KUKA KRL program: MyProgram_337().src

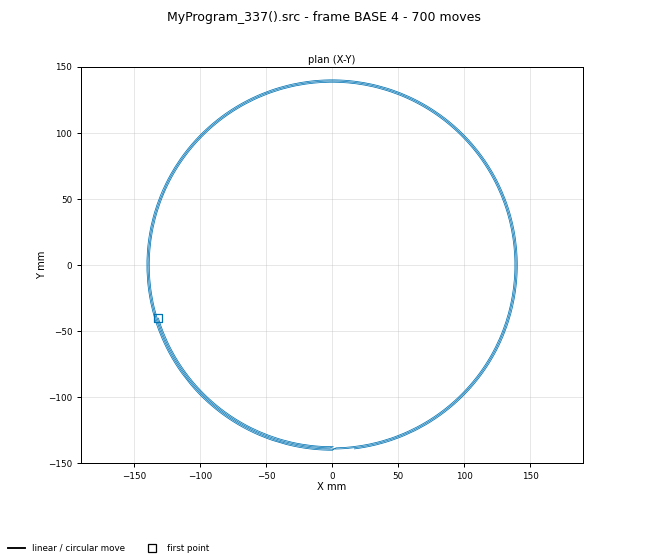
[picture p0: tool path of MyProgram_337().src in frame BASE 4, 700 of 700 moves have a stored position in this frame; points joined in program order, loops and branches not executed]
&ACCESS RVP
&REL 1
&PARAM TEMPLATE = C:\KRC\Roboter\Template\vorgabe
&PARAM EDITMASK = *
DEF MyProgram_337()
; ---- Setting reference (Base) ----
$BASE = BASE_DATA[4]

; --------------------------
; ---- Setting tool (TCP) ----
$TOOL = TOOL_DATA[3]
; --------------------------

$VEL.CP = VEL_APROX_PRINT
Startdeposition()
$VEL.CP = VEL_PRINT
LIN {X -131.5627,Y -40.1992,Z 190,A -156.4352,B 1.1423,C 0.1249,E1 0.9973,E2 249.9289} C_DIS
LIN {X -130.6707,Y -43.0129,Z 190,A -155.1283,B 1.1419,C 0.1281,E1 0.9985,E2 248.6121} C_DIS
LIN {X -129.6796,Y -45.9186,Z 190,A -153.4,B 1.1415,C 0.1315,E1 1.0001,E2 246.8238} C_DIS
LIN {X -127.8186,Y -50.8673,Z 190,A -150.9878,B 1.1409,C 0.1372,E1 1.0026,E2 244.3839} C_DIS
LIN {X -126.194,Y -54.7705,Z 190,A -149.1607,B 1.1403,C 0.1416,E1 1.0046,E2 242.5483} C_DIS
LIN {X -124.9534,Y -57.5445,Z 190,A -147.6737,B 1.14,C 0.1447,E1 1.0063,E2 241.0315} C_DIS
LIN {X -123.462,Y -60.6782,Z 190,A -146.0319,B 1.1395,C 0.1482,E1 1.0084,E2 239.3634} C_DIS
LIN {X -121.5451,Y -64.4341,Z 190,A -143.3556,B 1.139,C 0.1523,E1 1.0121,E2 236.5609} C_DIS
LIN {X -118.9555,Y -69.1002,Z 190,A -141.515,B 1.1383,C 0.1574,E1 1.0145,E2 234.7739} C_DIS
LIN {X -116.3723,Y -73.367,Z 190,A -139.2239,B 1.1376,C 0.162,E1 1.0179,E2 232.4537} C_DIS
LIN {X -113.9274,Y -77.1089,Z 190,A -137.1564,B 1.137,C 0.166,E1 1.0212,E2 230.3581} C_DIS
LIN {X -111.3595,Y -80.7731,Z 190,A -135.1136,B 1.1365,C 0.1699,E1 1.0245,E2 228.2907} C_DIS
LIN {X -108.6208,Y -84.4203,Z 190,A -132.998,B 1.1359,C 0.1736,E1 1.0282,E2 226.1454} C_DIS
LIN {X -105.7296,Y -88.0148,Z 190,A -130.861,B 1.1353,C 0.1773,E1 1.032,E2 223.9785} C_DIS
LIN {X -102.7599,Y -91.4648,Z 190,A -128.8416,B 1.1348,C 0.1808,E1 1.0358,E2 221.942} C_DIS
LIN {X -99.7983,Y -94.6873,Z 190,A -126.928,B 1.1343,C 0.1841,E1 1.0395,E2 220.0158} C_DIS
LIN {X -97.1901,Y -97.3623,Z 190,A -125.164,B 1.1338,C 0.1866,E1 1.043,E2 218.2226} C_DIS
LIN {X -94.7289,Y -99.7586,Z 190,A -123.479,B 1.1335,C 0.1888,E1 1.0465,E2 216.5018} C_DIS
LIN {X -90.9578,Y -103.2083,Z 190,A -121.3105,B 1.1329,C 0.1922,E1 1.0511,E2 214.3277} C_DIS
LIN {X -87.7491,Y -105.9496,Z 190,A -119.4335,B 1.1325,C 0.1947,E1 1.0552,E2 212.4338} C_DIS
LIN {X -84.3581,Y -108.669,Z 190,A -117.4741,B 1.1321,C 0.1972,E1 1.0595,E2 210.4532} C_DIS
LIN {X -80.6661,Y -111.4371,Z 190,A -115.4682,B 1.1316,C 0.1997,E1 1.0641,E2 208.4352} C_DIS
LIN {X -76.4637,Y -114.3615,Z 190,A -113.1651,B 1.1312,C 0.2022,E1 1.0695,E2 206.1076} C_DIS
LIN {X -72.9085,Y -116.6604,Z 190,A -111.1391,B 1.1309,C 0.2038,E1 1.0744,E2 204.0438} C_DIS
LIN {X -68.4116,Y -119.3531,Z 190,A -109.0245,B 1.1304,C 0.2063,E1 1.0795,E2 201.9387} C_DIS
LIN {X -64.6433,Y -121.4352,Z 190,A -107.1659,B 1.1301,C 0.208,E1 1.0842,E2 200.0705} C_DIS
LIN {X -61.1965,Y -123.2063,Z 190,A -105.6298,B 1.1298,C 0.2096,E1 1.088,E2 198.5452} C_DIS
LIN {X -57.9125,Y -124.7833,Z 190,A -104.2309,B 1.1295,C 0.2111,E1 1.0915,E2 197.1629} C_DIS
LIN {X -55.1219,Y -126.0421,Z 190,A -102.628,B 1.1295,C 0.2114,E1 1.0958,E2 195.5128} C_DIS
LIN {X -50.5791,Y -127.9339,Z 190,A -100.5694,B 1.1292,C 0.2128,E1 1.1011,E2 193.4524} C_DIS
LIN {X -47.9087,Y -128.9558,Z 190,A -99.21,B 1.1292,C 0.2132,E1 1.1048,E2 192.0684} C_DIS
LIN {X -43.7636,Y -130.4207,Z 190,A -97.4491,B 1.1289,C 0.2143,E1 1.1095,E2 190.3171} C_DIS
LIN {X -40.8951,Y -131.3497,Z 190,A -96.2332,B 1.1289,C 0.215,E1 1.1127,E2 189.1065} C_DIS
LIN {X -37.3559,Y -132.3985,Z 190,A -94.5915,B 1.1287,C 0.2153,E1 1.1172,E2 187.4493} C_DIS
LIN {X -33.9694,Y -133.3073,Z 190,A -93.1469,B 1.1287,C 0.2158,E1 1.1211,E2 186.0065} C_DIS
LIN {X -30.8122,Y -134.0724,Z 190,A -91.8493,B 1.1286,C 0.2163,E1 1.1247,E2 184.7163} C_DIS
LIN {X -26.9975,Y -134.8929,Z 190,A -89.6626,B 1.1288,C 0.2151,E1 1.1309,E2 182.4478} C_DIS
LIN {X -22.9337,Y -135.6426,Z 190,A -88.3319,B 1.1286,C 0.2163,E1 1.1345,E2 181.1729} C_DIS
LIN {X -16.4531,Y -136.5801,Z 190,A -85.5629,B 1.1286,C 0.2161,E1 1.1422,E2 178.3968} C_DIS
LIN {X -12.3209,Y -137.0166,Z 190,A -83.8051,B 1.1286,C 0.2158,E1 1.1472,E2 176.6343} C_DIS
LIN {X -8.3051,Y -137.3167,Z 190,A -82.2397,B 1.1286,C 0.2158,E1 1.1515,E2 175.0842} C_DIS
LIN {X -4.2325,Y -137.5031,Z 190,A -80.452,B 1.1288,C 0.2151,E1 1.1566,E2 173.2827} C_DIS
LIN {X 0.983,Y -137.5643,Z 190,A -78.8429,B 1.1286,C 0.2161,E1 1.1609,E2 171.7536} C_DIS
Enddeposition()
LIN {X 0.983,Y -137.5643,Z 190,A -78.843,B 1.1286,C 0.2161,E1 1.1609,E2 171.7538} C_DIS
Startdeposition()
$VEL.CP = VEL_PRINT
LIN {X -1.5333,Y -138.4601,Z 190,A -80.1965,B 1.1539,C 0.2192,E1 1.1826,E2 173.1713} C_DIS
LIN {X -4.6035,Y -138.392,Z 190,A -81.4508,B 1.1539,C 0.2195,E1 1.1791,E2 174.4239} C_DIS
LIN {X -8.8461,Y -138.184,Z 190,A -83.1886,B 1.1538,C 0.2199,E1 1.1742,E2 176.1597} C_DIS
LIN {X -12.4098,Y -137.9112,Z 190,A -84.6675,B 1.1538,C 0.2201,E1 1.17,E2 177.6394} C_DIS
LIN {X -15.5748,Y -137.5897,Z 190,A -85.981,B 1.1537,C 0.2202,E1 1.1663,E2 178.953} C_DIS
LIN {X -18.757,Y -137.1921,Z 190,A -87.3061,B 1.1537,C 0.2202,E1 1.1626,E2 180.2785} C_DIS
LIN {X -21.4733,Y -136.7914,Z 190,A -88.4926,B 1.1537,C 0.2204,E1 1.1593,E2 181.4726} C_DIS
LIN {X -25.1634,Y -136.1628,Z 190,A -90.0069,B 1.1537,C 0.2201,E1 1.1551,E2 182.9826} C_DIS
LIN {X -28.0039,Y -135.6054,Z 190,A -91.2463,B 1.1537,C 0.2201,E1 1.1517,E2 184.2285} C_DIS
LIN {X -31.6408,Y -134.8051,Z 190,A -92.7737,B 1.1538,C 0.2196,E1 1.1475,E2 185.7545} C_DIS
LIN {X -34.7188,Y -134.0445,Z 190,A -94.103,B 1.1538,C 0.2193,E1 1.1438,E2 187.0868} C_DIS
LIN {X -38.1008,Y -133.1236,Z 190,A -95.5818,B 1.154,C 0.2188,E1 1.1398,E2 188.5702} C_DIS
LIN {X -41.3291,Y -132.157,Z 190,A -97.0049,B 1.154,C 0.2183,E1 1.136,E2 189.9978} C_DIS
LIN {X -44.5521,Y -131.1056,Z 190,A -98.4415,B 1.1542,C 0.2176,E1 1.1321,E2 191.4398} C_DIS
LIN {X -47.7339,Y -129.9807,Z 190,A -99.8757,B 1.1543,C 0.2169,E1 1.1283,E2 192.8798} C_DIS
LIN {X -50.9696,Y -128.7465,Z 190,A -101.3517,B 1.1545,C 0.2161,E1 1.1244,E2 194.3623} C_DIS
LIN {X -54.0161,Y -127.4974,Z 190,A -102.7597,B 1.1546,C 0.2152,E1 1.1207,E2 195.7771} C_DIS
LIN {X -57.0709,Y -126.1589,Z 190,A -104.2036,B 1.1548,C 0.2142,E1 1.117,E2 197.2304} C_DIS
LIN {X -60.475,Y -124.5646,Z 190,A -105.8075,B 1.155,C 0.213,E1 1.1129,E2 198.8416} C_DIS
LIN {X -63.5979,Y -122.9995,Z 190,A -107.3149,B 1.1553,C 0.2118,E1 1.1091,E2 200.3582} C_DIS
LIN {X -66.31,Y -121.558,Z 190,A -108.7108,B 1.1555,C 0.2107,E1 1.1056,E2 201.7721} C_DIS
LIN {X -69.755,Y -119.6152,Z 190,A -110.3598,B 1.1558,C 0.209,E1 1.1015,E2 203.4232} C_DIS
LIN {X -72.6195,Y -117.8975,Z 190,A -111.8361,B 1.156,C 0.2076,E1 1.098,E2 204.913} C_DIS
LIN {X -76.1626,Y -115.64,Z 190,A -113.7142,B 1.1564,C 0.2057,E1 1.0935,E2 206.8112} C_DIS
LIN {X -79.8624,Y -113.1166,Z 190,A -115.672,B 1.1568,C 0.2035,E1 1.0889,E2 208.784} C_DIS
LIN {X -83.039,Y -110.8065,Z 190,A -117.3467,B 1.1571,C 0.2013,E1 1.0851,E2 210.4658} C_DIS
LIN {X -86.2373,Y -108.3351,Z 190,A -119.2008,B 1.1575,C 0.1991,E1 1.0809,E2 212.3457} C_DIS
LIN {X -89.3427,Y -105.7896,Z 190,A -120.9923,B 1.1579,C 0.1968,E1 1.077,E2 214.1555} C_DIS
LIN {X -92.7012,Y -102.8593,Z 190,A -122.8956,B 1.1584,C 0.1939,E1 1.073,E2 216.067} C_DIS
LIN {X -95.3316,Y -100.4262,Z 190,A -124.4946,B 1.1588,C 0.1915,E1 1.0697,E2 217.6824} C_DIS
LIN {X -97.9121,Y -97.9121,Z 190,A -126.1074,B 1.1592,C 0.1891,E1 1.0664,E2 219.3123} C_DIS
LIN {X -100.6879,Y -95.0542,Z 190,A -127.9781,B 1.1597,C 0.1863,E1 1.0628,E2 221.2139} C_DIS
LIN {X -103.4567,Y -92.034,Z 190,A -129.8673,B 1.1601,C 0.1833,E1 1.0592,E2 223.13} C_DIS
LIN {X -106.4321,Y -88.5758,Z 190,A -131.9282,B 1.1607,C 0.1797,E1 1.0554,E2 225.2148} C_DIS
LIN {X -109.1582,Y -85.1941,Z 190,A -133.7748,B 1.1612,C 0.1761,E1 1.0521,E2 227.0679} C_DIS
LIN {X -111.328,Y -82.3386,Z 190,A -135.4036,B 1.1617,C 0.1732,E1 1.0494,E2 228.7166} C_DIS
LIN {X -113.257,Y -79.6633,Z 190,A -136.9417,B 1.1621,C 0.1703,E1 1.0468,E2 230.2784} C_DIS
LIN {X -115.4099,Y -76.5122,Z 190,A -138.6491,B 1.1626,C 0.167,E1 1.0441,E2 232.0032} C_DIS
LIN {X -117.3303,Y -73.5334,Z 190,A -140.3787,B 1.163,C 0.1638,E1 1.0415,E2 233.7687} C_DIS
LIN {X -119.6061,Y -69.7705,Z 190,A -142.2935,B 1.1636,C 0.1597,E1 1.0387,E2 235.6961} C_DIS
LIN {X -121.3495,Y -66.6923,Z 190,A -143.9218,B 1.1641,C 0.1563,E1 1.0365,E2 237.3465} C_DIS
LIN {X -122.9093,Y -63.7697,Z 190,A -145.4555,B 1.1645,C 0.1531,E1 1.0344,E2 238.9021} C_DIS
LIN {X -124.3492,Y -60.9117,Z 190,A -146.9699,B 1.1649,C 0.1499,E1 1.0325,E2 240.442} C_DIS
LIN {X -126.0443,Y -57.3271,Z 190,A -148.7649,B 1.1654,C 0.1459,E1 1.0304,E2 242.2575} C_DIS
LIN {X -127.4383,Y -54.1575,Z 190,A -150.3709,B 1.1659,C 0.1424,E1 1.0286,E2 243.8864} C_DIS
LIN {X -128.7334,Y -51.0022,Z 190,A -151.9557,B 1.1663,C 0.1388,E1 1.0269,E2 245.4942} C_DIS
LIN {X -129.9689,Y -47.7667,Z 190,A -153.5679,B 1.1667,C 0.1351,E1 1.0253,E2 247.13} C_DIS
LIN {X -131.0942,Y -44.585,Z 190,A -155.1384,B 1.1671,C 0.1315,E1 1.0238,E2 248.7233} C_DIS
LIN {X -132.157,Y -41.3291,Z 190,A -156.7397,B 1.1676,C 0.1277,E1 1.0224,E2 250.3487} C_DIS
LIN {X -132.9702,Y -38.6248,Z 190,A -158.0672,B 1.1679,C 0.1246,E1 1.0214,E2 251.6969} C_DIS
LIN {X -133.9972,Y -34.9033,Z 190,A -159.8584,B 1.1683,C 0.1203,E1 1.02,E2 253.5133} C_DIS
LIN {X -134.6974,Y -32.0879,Z 190,A -161.233,B 1.1687,C 0.117,E1 1.0191,E2 254.9104} C_DIS
LIN {X -135.4719,Y -28.6461,Z 190,A -162.8891,B 1.1691,C 0.113,E1 1.0181,E2 256.5918} C_DIS
LIN {X -136.135,Y -25.311,Z 190,A -164.4774,B 1.1694,C 0.1091,E1 1.0173,E2 258.2034} C_DIS
LIN {X -136.7119,Y -21.9868,Z 190,A -166.0584,B 1.1698,C 0.1052,E1 1.0165,E2 259.8081} C_DIS
LIN {X -137.3216,Y -17.7691,Z 190,A -168.1258,B 1.1702,C 0.1002,E1 1.0157,E2 261.9143} C_DIS
LIN {X -137.7568,Y -14.0223,Z 190,A -169.8359,B 1.1706,C 0.0958,E1 1.0152,E2 263.6432} C_DIS
LIN {X -138.0416,Y -10.8667,Z 190,A -171.3266,B 1.1709,C 0.0921,E1 1.0148,E2 265.1566} C_DIS
LIN {X -138.2526,Y -7.7319,Z 190,A -172.8055,B 1.1712,C 0.0884,E1 1.0146,E2 266.658} C_DIS
LIN {X -138.3726,Y -5.1056,Z 190,A -174.0489,B 1.1714,C 0.0853,E1 1.0144,E2 267.9209} C_DIS
LIN {X -138.4596,Y -1.5648,Z 190,A -175.7119,B 1.1717,C 0.0811,E1 1.0144,E2 269.6085} C_DIS
LIN {X -138.4606,Y 1.4676,Z 190,A -177.1471,B 1.172,C 0.0775,E1 1.0144,E2 271.0662} C_DIS
LIN {X -138.3915,Y 4.6201,Z 190,A -178.6333,B 1.1722,C 0.0737,E1 1.0144,E2 272.5749} C_DIS
LIN {X -138.2526,Y 7.7319,Z 190,A 179.8943,B 1.1724,C 0.0701,E1 1.0147,E2 274.0701} C_DIS
LIN {X -137.9596,Y 11.8371,Z 190,A 177.8799,B 1.1727,C 0.0651,E1 1.0151,E2 276.1229} C_DIS
LIN {X -137.5897,Y 15.5748,Z 190,A 176.1754,B 1.1729,C 0.0607,E1 1.0156,E2 277.8456} C_DIS
LIN {X -137.1921,Y 18.757,Z 190,A 174.6616,B 1.1731,C 0.057,E1 1.0162,E2 279.3821} C_DIS
LIN {X -136.7119,Y 21.9868,Z 190,A 173.1212,B 1.1733,C 0.0531,E1 1.0168,E2 280.9455} C_DIS
LIN {X -136.222,Y 24.8327,Z 190,A 171.7669,B 1.1735,C 0.0498,E1 1.0175,E2 282.319} C_DIS
LIN {X -135.5217,Y 28.4151,Z 190,A 170.0405,B 1.1736,C 0.0456,E1 1.0185,E2 284.0714} C_DIS
LIN {X -134.8051,Y 31.6408,Z 190,A 168.4855,B 1.1738,C 0.0418,E1 1.0195,E2 285.6489} C_DIS
LIN {X -134.0144,Y 34.8374,Z 190,A 166.9367,B 1.1739,C 0.038,E1 1.0205,E2 287.22} C_DIS
LIN {X -133.2721,Y 37.5697,Z 190,A 165.6011,B 1.174,C 0.0348,E1 1.0216,E2 288.5749} C_DIS
LIN {X -132.157,Y 41.3291,Z 190,A 163.7687,B 1.1741,C 0.0304,E1 1.0231,E2 290.4322} C_DIS
LIN {X -131.1056,Y 44.5521,Z 190,A 162.1808,B 1.1742,C 0.0267,E1 1.0245,E2 292.0419} C_DIS
LIN {X -130.095,Y 47.4168,Z 190,A 160.7715,B 1.1742,C 0.0234,E1 1.0258,E2 293.4689} C_DIS
LIN {X -128.8741,Y 50.6414,Z 190,A 159.1246,B 1.1744,C 0.0196,E1 1.0275,E2 295.1416} C_DIS
LIN {X -127.4383,Y 54.1575,Z 190,A 157.3795,B 1.1744,C 0.0156,E1 1.0294,E2 296.9069} C_DIS
LIN {X -126.0443,Y 57.3271,Z 190,A 155.7686,B 1.1744,C 0.012,E1 1.0313,E2 298.5384} C_DIS
LIN {X -124.5646,Y 60.475,Z 190,A 154.1532,B 1.1744,C 0.0084,E1 1.0332,E2 300.174} C_DIS
LIN {X -122.9995,Y 63.5979,Z 190,A 152.5345,B 1.1745,C 0.0049,E1 1.0353,E2 301.8125} C_DIS
LIN {X -121.3617,Y 66.6699,Z 190,A 150.9217,B 1.1745,C 0.0014,E1 1.0375,E2 303.4449} C_DIS
LIN {X -119.6152,Y 69.755,Z 190,A 149.2906,B 1.1745,C -0.002,E1 1.0398,E2 305.0947} C_DIS
LIN {X -117.6028,Y 73.0955,Z 190,A 147.4279,B 1.1745,C -0.0057,E1 1.0426,E2 306.9857} C_DIS
LIN {X -115.4099,Y 76.5122,Z 190,A 145.6313,B 1.1745,C -0.0094,E1 1.0453,E2 308.7951} C_DIS
LIN {X -113.4086,Y 79.4483,Z 190,A 144.0046,B 1.1745,C -0.0126,E1 1.0479,E2 310.4392} C_DIS
LIN {X -111.3388,Y 82.3239,Z 190,A 142.3848,B 1.1745,C -0.0157,E1 1.0507,E2 312.0761} C_DIS
LIN {X -108.8631,Y 85.5697,Z 190,A 140.465,B 1.1744,C -0.0192,E1 1.054,E2 314.0217} C_DIS
LIN {X -106.3646,Y 88.6574,Z 190,A 138.7225,B 1.1744,C -0.0224,E1 1.0571,E2 315.7747} C_DIS
LIN {X -104.0496,Y 91.3631,Z 190,A 137.1107,B 1.1742,C -0.0253,E1 1.0601,E2 317.4016} C_DIS
LIN {X -101.6514,Y 94.0241,Z 190,A 135.4942,B 1.1742,C -0.028,E1 1.0632,E2 319.0328} C_DIS
LIN {X -99.1712,Y 96.6366,Z 190,A 133.7491,B 1.1742,C -0.0306,E1 1.0666,E2 320.8063} C_DIS
LIN {X -95.9927,Y 99.7946,Z 190,A 131.8639,B 1.174,C -0.0339,E1 1.0704,E2 322.6938} C_DIS
LIN {X -93.3781,Y 102.2453,Z 190,A 130.2623,B 1.174,C -0.0363,E1 1.0738,E2 324.3082} C_DIS
LIN {X -90.7025,Y 104.6261,Z 190,A 128.6684,B 1.1739,C -0.0387,E1 1.0771,E2 325.914} C_DIS
LIN {X -87.7038,Y 107.1514,Z 190,A 126.8337,B 1.1739,C -0.041,E1 1.0812,E2 327.7719} C_DIS
LIN {X -84.4742,Y 109.7163,Z 190,A 125.1008,B 1.1737,C -0.0435,E1 1.085,E2 329.5067} C_DIS
LIN {X -81.8311,Y 111.7008,Z 190,A 123.6073,B 1.1737,C -0.0454,E1 1.0884,E2 331.0137} C_DIS
LIN {X -78.7334,Y 113.9061,Z 190,A 121.8818,B 1.1736,C -0.0473,E1 1.0924,E2 332.7555} C_DIS
LIN {X -75.0431,Y 116.3704,Z 190,A 120.0271,B 1.1735,C -0.0496,E1 1.0968,E2 334.6112} C_DIS
LIN {X -72.0291,Y 118.2598,Z 190,A 118.4772,B 1.1735,C -0.0513,E1 1.1005,E2 336.169} C_DIS
LIN {X -69.0081,Y 120.0476,Z 190,A 116.9506,B 1.1733,C -0.0528,E1 1.1042,E2 337.7031} C_DIS
LIN {X -65.5833,Y 121.9516,Z 190,A 115.1729,B 1.1733,C -0.0543,E1 1.1087,E2 339.4974} C_DIS
LIN {X -62.0716,Y 123.7765,Z 190,A 113.5443,B 1.1732,C -0.0559,E1 1.1127,E2 341.1241} C_DIS
LIN {X -59.317,Y 125.1178,Z 190,A 112.1891,B 1.1732,C -0.0569,E1 1.1162,E2 342.4883} C_DIS
LIN {X -55.7771,Y 126.7376,Z 190,A 110.5613,B 1.1731,C -0.0582,E1 1.1204,E2 344.1172} C_DIS
LIN {X -52.5981,Y 128.0896,Z 190,A 109.0846,B 1.1731,C -0.0592,E1 1.1242,E2 345.5984} C_DIS
LIN {X -49.7256,Y 129.2301,Z 190,A 107.7366,B 1.173,C -0.06,E1 1.1278,E2 346.9533} C_DIS
LIN {X -46.1606,Y 130.5479,Z 190,A 106.1491,B 1.173,C -0.0609,E1 1.132,E2 348.5418} C_DIS
LIN {X -42.9743,Y 131.631,Z 190,A 104.7275,B 1.173,C -0.0616,E1 1.1358,E2 349.9658} C_DIS
LIN {X -40.0982,Y 132.5337,Z 190,A 103.4263,B 1.1729,C -0.0621,E1 1.1393,E2 351.2724} C_DIS
LIN {X -36.5186,Y 133.5661,Z 190,A 101.8861,B 1.1729,C -0.0627,E1 1.1435,E2 352.8117} C_DIS
LIN {X -33.2553,Y 134.416,Z 190,A 100.472,B 1.1729,C -0.0631,E1 1.1474,E2 354.2273} C_DIS
LIN {X -30.0602,Y 135.1662,Z 190,A 99.1004,B 1.1729,C -0.0634,E1 1.1511,E2 355.5997} C_DIS
LIN {X -27.3307,Y 135.7424,Z 190,A 97.8913,B 1.1729,C -0.0636,E1 1.1545,E2 356.8142} C_DIS
LIN {X -23.5901,Y 136.4444,Z 190,A 96.3567,B 1.1728,C -0.0638,E1 1.1587,E2 358.3437} C_DIS
LIN {X -20.4192,Y 136.9546,Z 190,A 95.0264,B 1.1728,C -0.0639,E1 1.1624,E2 359.6736} C_DIS
LIN {X -17.1963,Y 137.3967,Z 190,A 93.6834,B 1.1728,C -0.0639,E1 1.1662,E2 361.0156} C_DIS
LIN {X -14.0223,Y 137.7568,Z 190,A 92.3682,B 1.1728,C -0.0639,E1 1.1699,E2 362.3295} C_DIS
LIN {X -11.3116,Y 138.004,Z 190,A 91.2148,B 1.1728,C -0.0636,E1 1.1731,E2 363.4853} C_DIS
LIN {X -7.7319,Y 138.2526,Z 190,A 89.7813,B 1.1728,C -0.0634,E1 1.1771,E2 364.9127} C_DIS
LIN {X -4.6518,Y 138.3903,Z 190,A 88.5296,B 1.1728,C -0.0632,E1 1.1807,E2 366.1611} C_DIS
LIN {X -1.5648,Y 138.4596,Z 190,A 87.2658,B 1.1728,C -0.0628,E1 1.1842,E2 367.4229} C_DIS
LIN {X 1.5333,Y 138.4601,Z 190,A 86.0037,B 1.1728,C -0.0624,E1 1.1878,E2 368.6823} C_DIS
LIN {X 5.9375,Y 138.3401,Z 190,A 84.2014,B 1.1729,C -0.0616,E1 1.1928,E2 370.4815} C_DIS
LIN {X 9.2646,Y 138.1582,Z 190,A 82.8632,B 1.1729,C -0.0609,E1 1.1966,E2 371.8148} C_DIS
LIN {X 12.4098,Y 137.9112,Z 190,A 81.5888,B 1.1729,C -0.0603,E1 1.2001,E2 373.0852} C_DIS
LIN {X 15.5748,Y 137.5897,Z 190,A 80.3071,B 1.173,C -0.0595,E1 1.2037,E2 374.3626} C_DIS
LIN {X 18.3167,Y 137.2498,Z 190,A 79.1591,B 1.173,C -0.0587,E1 1.2069,E2 375.5107} C_DIS
LIN {X 21.7804,Y 136.7438,Z 190,A 77.7858,B 1.1731,C -0.0578,E1 1.2107,E2 376.8752} C_DIS
LIN {X 24.7849,Y 136.2305,Z 190,A 76.5437,B 1.1731,C -0.0568,E1 1.2142,E2 378.1147} C_DIS
LIN {X 28.4151,Y 135.5217,Z 190,A 75.1,B 1.1732,C -0.0557,E1 1.2181,E2 379.5483} C_DIS
LIN {X 31.0138,Y 134.9483,Z 190,A 74.022,B 1.1732,C -0.0547,E1 1.2211,E2 380.6233} C_DIS
LIN {X 34.8374,Y 134.0144,Z 190,A 72.4791,B 1.1733,C -0.0533,E1 1.2253,E2 382.1562} C_DIS
LIN {X 38.1008,Y 133.1236,Z 190,A 71.1409,B 1.1733,C -0.052,E1 1.2289,E2 383.4871} C_DIS
LIN {X 41.0793,Y 132.2334,Z 190,A 69.9279,B 1.1734,C -0.0508,E1 1.2321,E2 384.6914} C_DIS
LIN {X 44.5521,Y 131.1056,Z 190,A 68.4767,B 1.1734,C -0.0492,E1 1.236,E2 386.1356} C_DIS
LIN {X 47.7339,Y 129.9807,Z 190,A 67.1514,B 1.1736,C -0.0477,E1 1.2395,E2 387.4525} C_DIS
LIN {X 50.4491,Y 128.9488,Z 190,A 66.0118,B 1.1736,C -0.0464,E1 1.2424,E2 388.5847} C_DIS
LIN {X 53.6927,Y 127.6324,Z 190,A 64.6068,B 1.1736,C -0.0446,E1 1.2461,E2 389.9845} C_DIS
LIN {X 56.8457,Y 126.2596,Z 190,A 63.2922,B 1.1737,C -0.043,E1 1.2494,E2 391.2865} C_DIS
LIN {X 60.475,Y 124.5646,Z 190,A 61.7449,B 1.1738,C -0.0409,E1 1.2533,E2 392.821} C_DIS
LIN {X 63.3828,Y 123.109,Z 190,A 60.4741,B 1.1738,C -0.0392,E1 1.2565,E2 394.083} C_DIS
LIN {X 66.6766,Y 121.358,Z 190,A 59.037,B 1.1739,C -0.0371,E1 1.26,E2 395.5078} C_DIS
LIN {X 70.1625,Y 119.3758,Z 190,A 57.4364,B 1.174,C -0.0346,E1 1.2639,E2 397.1015} C_DIS
LIN {X 73.8304,Y 117.1428,Z 190,A 55.7531,B 1.174,C -0.032,E1 1.2679,E2 398.7738} C_DIS
LIN {X 77.7577,Y 114.5737,Z 190,A 53.9986,B 1.1742,C -0.0293,E1 1.2719,E2 400.5066} C_DIS
LIN {X 80.8518,Y 112.4122,Z 190,A 52.606,B 1.1742,C -0.0272,E1 1.2751,E2 401.8794} C_DIS
LIN {X 83.7509,Y 110.2693,Z 190,A 51.2056,B 1.1742,C -0.0248,E1 1.2782,E2 403.2692} C_DIS
LIN {X 86.5809,Y 108.0616,Z 190,A 49.8354,B 1.1743,C -0.0224,E1 1.2812,E2 404.6259} C_DIS
LIN {X 89.6037,Y 105.5677,Z 190,A 48.2648,B 1.1743,C -0.0194,E1 1.2845,E2 406.1906} C_DIS
LIN {X 92.7012,Y 102.8593,Z 190,A 46.7776,B 1.1743,C -0.0169,E1 1.2876,E2 407.6526} C_DIS
LIN {X 95.3316,Y 100.4262,Z 190,A 45.4179,B 1.1744,C -0.0144,E1 1.2904,E2 408.9978} C_DIS
LIN {X 97.8714,Y 97.9525,Z 190,A 43.9955,B 1.1744,C -0.0115,E1 1.2932,E2 410.4151} C_DIS
LIN {X 101.0285,Y 94.6932,Z 190,A 42.3587,B 1.1744,C -0.0085,E1 1.2963,E2 412.0235} C_DIS
LIN {X 103.4446,Y 92.0477,Z 190,A 40.9416,B 1.1745,C -0.0055,E1 1.2989,E2 413.433} C_DIS
LIN {X 106.3528,Y 88.6714,Z 190,A 39.3276,B 1.1745,C -0.0025,E1 1.3018,E2 415.0198} C_DIS
LIN {X 108.6065,Y 85.8963,Z 190,A 37.9813,B 1.1745,C 0.0003,E1 1.3042,E2 416.3504} C_DIS
LIN {X 110.7956,Y 83.0536,Z 190,A 36.5496,B 1.1745,C 0.0035,E1 1.3066,E2 417.776} C_DIS
LIN {X 113.4086,Y 79.4483,Z 190,A 34.9668,B 1.1745,C 0.0066,E1 1.3091,E2 419.3279} C_DIS
LIN {X 115.641,Y 76.1612,Z 190,A 33.4168,B 1.1745,C 0.0101,E1 1.3115,E2 420.8669} C_DIS
LIN {X 117.7976,Y 72.7824,Z 190,A 31.8894,B 1.1745,C 0.0135,E1 1.3137,E2 422.3787} C_DIS
LIN {X 120.0476,Y 69.0081,Z 190,A 30.3377,B 1.1745,C 0.0166,E1 1.3159,E2 423.8985} C_DIS
LIN {X 122.0218,Y 65.4527,Z 190,A 28.7953,B 1.1743,C 0.0201,E1 1.3179,E2 425.4242} C_DIS
LIN {X 123.7765,Y 62.0716,Z 190,A 27.4023,B 1.1743,C 0.0232,E1 1.3197,E2 426.7952} C_DIS
LIN {X 125.2998,Y 58.936,Z 190,A 26.1062,B 1.1743,C 0.0261,E1 1.3212,E2 428.0736} C_DIS
LIN {X 126.7376,Y 55.7771,Z 190,A 24.8166,B 1.1742,C 0.0291,E1 1.3227,E2 429.3456} C_DIS
LIN {X 127.9617,Y 52.9044,Z 190,A 23.6625,B 1.1741,C 0.0317,E1 1.3239,E2 430.483} C_DIS
LIN {X 129.3557,Y 49.4025,Z 190,A 22.2552,B 1.1741,C 0.035,E1 1.3253,E2 431.8719} C_DIS
LIN {X 130.3722,Y 46.6479,Z 190,A 21.1444,B 1.1739,C 0.0377,E1 1.3264,E2 432.9702} C_DIS
LIN {X 131.584,Y 43.1152,Z 190,A 19.7764,B 1.1739,C 0.0408,E1 1.3276,E2 434.3166} C_DIS
LIN {X 132.6408,Y 39.7483,Z 190,A 18.4755,B 1.1737,C 0.0439,E1 1.3286,E2 435.5982} C_DIS
LIN {X 133.5661,Y 36.5186,Z 190,A 17.2381,B 1.1736,C 0.0468,E1 1.3295,E2 436.817} C_DIS
LIN {X 134.2946,Y 33.7335,Z 190,A 16.1541,B 1.1735,C 0.0495,E1 1.3303,E2 437.888} C_DIS
LIN {X 135.1662,Y 30.0602,Z 190,A 14.7703,B 1.1733,C 0.0527,E1 1.3311,E2 439.25} C_DIS
LIN {X 135.7957,Y 27.0688,Z 190,A 13.6299,B 1.1733,C 0.0555,E1 1.3318,E2 440.3752} C_DIS
LIN {X 136.4444,Y 23.5901,Z 190,A 12.333,B 1.1731,C 0.0586,E1 1.3324,E2 441.6515} C_DIS
LIN {X 136.9546,Y 20.4192,Z 190,A 11.1508,B 1.1729,C 0.0615,E1 1.3329,E2 442.8156} C_DIS
LIN {X 137.3967,Y 17.1963,Z 190,A 9.9456,B 1.1728,C 0.0644,E1 1.3333,E2 444.0035} C_DIS
LIN {X 137.7568,Y 14.0223,Z 190,A 8.7664,B 1.1726,C 0.0673,E1 1.3337,E2 445.1651} C_DIS
LIN {X 138.0416,Y 10.8667,Z 190,A 7.5971,B 1.1724,C 0.0701,E1 1.334,E2 446.3169} C_DIS
LIN {X 138.2526,Y 7.7319,Z 190,A 6.4376,B 1.1723,C 0.0729,E1 1.3342,E2 447.4589} C_DIS
LIN {X 138.4336,Y 3.105,Z 190,A 4.7291,B 1.172,C 0.0771,E1 1.3343,E2 449.1417} C_DIS
LIN {X 138.4686,Y 0,Z 190,A 3.5732,B 1.1718,C 0.0799,E1 1.3343,E2 450.2816} C_DIS
LIN {X 138.4409,Y -2.687,Z 190,A 2.5616,B 1.1716,C 0.0825,E1 1.3343,E2 451.2807} C_DIS
LIN {X 138.331,Y -6.173,Z 190,A 1.2952,B 1.1714,C 0.0855,E1 1.3342,E2 452.525} C_DIS
LIN {X 138.0657,Y -10.5359,Z 190,A -0.3229,B 1.1711,C 0.0894,E1 1.3339,E2 454.1192} C_DIS
LIN {X 137.7599,Y -13.99,Z 190,A -1.6091,B 1.1709,C 0.0925,E1 1.3335,E2 455.3868} C_DIS
LIN {X 137.4006,Y -17.1639,Z 190,A -2.7928,B 1.1706,C 0.0954,E1 1.3332,E2 456.5532} C_DIS
LIN {X 136.9643,Y -20.3539,Z 190,A -3.9866,B 1.1704,C 0.0983,E1 1.3327,E2 457.7296} C_DIS
LIN {X 136.466,Y -23.4605,Z 190,A -5.1388,B 1.1702,C 0.101,E1 1.3322,E2 458.8629} C_DIS
LIN {X 135.8494,Y -26.8046,Z 190,A -6.4138,B 1.1699,C 0.1042,E1 1.3315,E2 460.1213} C_DIS
LIN {X 135.1737,Y -30.0273,Z 190,A -7.6354,B 1.1696,C 0.1071,E1 1.3308,E2 461.3251} C_DIS
LIN {X 134.4239,Y -33.2223,Z 190,A -8.8503,B 1.1694,C 0.11,E1 1.33,E2 462.5218} C_DIS
LIN {X 133.6047,Y -36.3752,Z 190,A -10.065,B 1.1691,C 0.1129,E1 1.3292,E2 463.7197} C_DIS
LIN {X 132.6508,Y -39.7154,Z 190,A -11.3531,B 1.1688,C 0.1159,E1 1.3282,E2 464.9889} C_DIS
LIN {X 131.6524,Y -42.9085,Z 190,A -12.5963,B 1.1685,C 0.1188,E1 1.3271,E2 466.214} C_DIS
LIN {X 130.5479,Y -46.1606,Z 190,A -13.8739,B 1.1682,C 0.1218,E1 1.326,E2 467.4734} C_DIS
LIN {X 129.5642,Y -48.847,Z 190,A -14.943,B 1.1679,C 0.1243,E1 1.3249,E2 468.5278} C_DIS
LIN {X 128.1032,Y -52.5656,Z 190,A -16.4263,B 1.1676,C 0.1277,E1 1.3234,E2 469.9895} C_DIS
LIN {X 126.7661,Y -55.7124,Z 190,A -17.7005,B 1.1672,C 0.1306,E1 1.322,E2 471.2457} C_DIS
LIN {X 125.33,Y -58.8718,Z 190,A -18.994,B 1.1669,C 0.1335,E1 1.3205,E2 472.5209} C_DIS
LIN {X 123.875,Y -61.8729,Z 190,A -20.2434,B 1.1666,C 0.1363,E1 1.319,E2 473.7536} C_DIS
LIN {X 121.7784,Y -65.9058,Z 190,A -21.9379,B 1.1661,C 0.14,E1 1.3168,E2 475.424} C_DIS
LIN {X 120.0566,Y -68.9925,Z 190,A -23.2598,B 1.1658,C 0.1429,E1 1.315,E2 476.7279} C_DIS
LIN {X 118.2691,Y -72.0136,Z 190,A -24.5743,B 1.1654,C 0.1457,E1 1.3132,E2 478.0245} C_DIS
LIN {X 116.1802,Y -75.3362,Z 190,A -26.1146,B 1.165,C 0.1493,E1 1.3109,E2 479.5546} C_DIS
LIN {X 113.9165,Y -78.7185,Z 190,A -27.5717,B 1.1646,C 0.1521,E1 1.3086,E2 480.9818} C_DIS
LIN {X 111.8662,Y -81.6058,Z 190,A -28.9041,B 1.1643,C 0.1548,E1 1.3065,E2 482.2969} C_DIS
LIN {X 109.7274,Y -84.4597,Z 190,A -30.3414,B 1.1638,C 0.1581,E1 1.3041,E2 483.7301} C_DIS
LIN {X 106.8889,Y -88.0242,Z 190,A -32.0609,B 1.1634,C 0.1615,E1 1.3011,E2 485.4281} C_DIS
LIN {X 104.0496,Y -91.3631,Z 190,A -33.6175,B 1.163,C 0.1642,E1 1.2983,E2 486.9505} C_DIS
LIN {X 101.6514,Y -94.0241,Z 190,A -35.0721,B 1.1625,C 0.1674,E1 1.2955,E2 488.4024} C_DIS
LIN {X 98.6316,Y -97.1868,Z 190,A -36.7006,B 1.1621,C 0.1703,E1 1.2924,E2 490.0071} C_DIS
LIN {X 95.5537,Y -100.2141,Z 190,A -38.2996,B 1.1617,C 0.1731,E1 1.2892,E2 491.5813} C_DIS
LIN {X 92.7283,Y -102.8348,Z 190,A -39.7321,B 1.1613,C 0.1756,E1 1.2863,E2 492.9924} C_DIS
LIN {X 90.0382,Y -105.1982,Z 190,A -41.1893,B 1.1609,C 0.1785,E1 1.2832,E2 494.4473} C_DIS
LIN {X 86.5809,Y -108.0616,Z 190,A -42.8861,B 1.1604,C 0.1813,E1 1.2796,E2 496.123} C_DIS
LIN {X 83.0536,Y -110.7956,Z 190,A -44.5128,B 1.1601,C 0.1837,E1 1.276,E2 497.7202} C_DIS
LIN {X 80.1753,Y -112.8959,Z 190,A -45.8764,B 1.1597,C 0.1859,E1 1.2729,E2 499.0693} C_DIS
LIN {X 77.2504,Y -114.9171,Z 190,A -47.2379,B 1.1594,C 0.188,E1 1.2698,E2 500.4164} C_DIS
LIN {X 74.0364,Y -117.0128,Z 190,A -48.8055,B 1.1589,C 0.1907,E1 1.2661,E2 501.9824} C_DIS
LIN {X 70.5153,Y -119.1686,Z 190,A -50.3084,B 1.1586,C 0.1926,E1 1.2626,E2 503.4575} C_DIS
LIN {X 67.4768,Y -120.915,Z 190,A -51.6652,B 1.1583,C 0.1946,E1 1.2593,E2 504.8022} C_DIS
LIN {X 64.0128,Y -122.7816,Z 190,A -53.2094,B 1.1579,C 0.1968,E1 1.2555,E2 506.3356} C_DIS
LIN {X 60.507,Y -124.5488,Z 190,A -54.7105,B 1.1576,C 0.1987,E1 1.2517,E2 507.8203} C_DIS
LIN {X 57.7082,Y -125.8681,Z 190,A -55.9394,B 1.1573,C 0.2003,E1 1.2486,E2 509.0428} C_DIS
LIN {X 54.1575,Y -127.4383,Z 190,A -57.4267,B 1.157,C 0.202,E1 1.2448,E2 510.5143} C_DIS
LIN {X 51.0022,Y -128.7334,Z 190,A -58.7569,B 1.1567,C 0.2036,E1 1.2414,E2 511.8339} C_DIS
LIN {X 48.1583,Y -129.8222,Z 190,A -59.9791,B 1.1565,C 0.2051,E1 1.2382,E2 513.0516} C_DIS
LIN {X 44.585,Y -131.0942,Z 190,A -61.4393,B 1.1562,C 0.2065,E1 1.2343,E2 514.4973} C_DIS
LIN {X 41.3291,Y -132.157,Z 190,A -62.7866,B 1.156,C 0.2079,E1 1.2308,E2 515.8355} C_DIS
LIN {X 38.5206,Y -133.0007,Z 190,A -63.9344,B 1.1558,C 0.209,E1 1.2277,E2 516.9747} C_DIS
LIN {X 34.9033,Y -133.9972,Z 190,A -65.4249,B 1.1555,C 0.2104,E1 1.2236,E2 518.4573} C_DIS
LIN {X 31.6408,Y -134.8051,Z 190,A -66.7559,B 1.1553,C 0.2115,E1 1.22,E2 519.7807} C_DIS
LIN {X 28.448,Y -135.5146,Z 190,A -68.0546,B 1.1551,C 0.2126,E1 1.2165,E2 521.0724} C_DIS
LIN {X 25.229,Y -136.1507,Z 190,A -69.358,B 1.1549,C 0.2136,E1 1.2129,E2 522.3689} C_DIS
LIN {X 22.5041,Y -136.6256,Z 190,A -70.5057,B 1.1548,C 0.2145,E1 1.2097,E2 523.5177} C_DIS
LIN {X 18.7896,Y -137.1879,Z 190,A -71.9661,B 1.1546,C 0.2154,E1 1.2057,E2 524.9656} C_DIS
LIN {X 15.6071,Y -137.5863,Z 190,A -73.2521,B 1.1545,C 0.2162,E1 1.2021,E2 526.2464} C_DIS
LIN {X 12.442,Y -137.9085,Z 190,A -74.5306,B 1.1543,C 0.2169,E1 1.1985,E2 527.5202} C_DIS
LIN {X 9.6268,Y -138.1321,Z 190,A -75.6434,B 1.1543,C 0.2174,E1 1.1954,E2 528.6256} C_DIS
LIN {X 6.347,Y -138.3222,Z 190,A -77.0003,B 1.1541,C 0.2181,E1 1.1916,E2 529.983} C_DIS
LIN {X 3.105,Y -138.4336,Z 190,A -78.3088,B 1.1541,C 0.2186,E1 1.1879,E2 531.2873} C_DIS
LIN {X 3.105,Y -138.4336,Z 190,A -78.3088,B 1.1541,C 0.2186,E1 1.1879,E2 531.2873} C_DIS
Enddeposition()
LIN {X 0.9972,Y -139.3583,Z 190,A -78.8814,B 1.1793,C 0.2196,E1 1.2117,E2 531.8356} C_DIS
Startdeposition()
$VEL.CP = VEL_PRINT
LIN {X 4.5028,Y -139.294,Z 190,A -77.3131,B 1.1795,C 0.2185,E1 1.2161,E2 530.2481} C_DIS
LIN {X 8.4891,Y -139.1065,Z 190,A -75.6663,B 1.1797,C 0.2177,E1 1.2208,E2 528.5995} C_DIS
LIN {X 12.0274,Y -138.8456,Z 190,A -74.2951,B 1.1798,C 0.2171,E1 1.2246,E2 527.2402} C_DIS
LIN {X 15.8039,Y -138.468,Z 190,A -72.8065,B 1.1799,C 0.2164,E1 1.2287,E2 525.7611} C_DIS
LIN {X 18.2881,Y -138.1602,Z 190,A -71.7774,B 1.1801,C 0.2156,E1 1.2316,E2 524.7314} C_DIS
LIN {X 21.6643,Y -137.6714,Z 190,A -70.4202,B 1.1802,C 0.2147,E1 1.2354,E2 523.38} C_DIS
LIN {X 25.3643,Y -137.04,Z 190,A -68.4345,B 1.1808,C 0.2116,E1 1.2411,E2 521.3288} C_DIS
LIN {X 29.5933,Y -136.187,Z 190,A -67.1716,B 1.1808,C 0.2121,E1 1.2443,E2 520.1392} C_DIS
LIN {X 33.6369,Y -135.2465,Z 190,A -65.4353,B 1.1811,C 0.2102,E1 1.2491,E2 518.3977} C_DIS
LIN {X 37.8045,Y -134.1398,Z 190,A -63.903,B 1.1812,C 0.2094,E1 1.2532,E2 516.899} C_DIS
LIN {X 41.2567,Y -133.1192,Z 190,A -62.4079,B 1.1815,C 0.2076,E1 1.2572,E2 515.4008} C_DIS
LIN {X 44.296,Y -132.1383,Z 190,A -61.2043,B 1.1817,C 0.2065,E1 1.2604,E2 514.2121} C_DIS
LIN {X 47.5321,Y -131.009,Z 190,A -59.8432,B 1.182,C 0.205,E1 1.264,E2 512.8571} C_DIS
LIN {X 51.1616,Y -129.6363,Z 190,A -58.3681,B 1.1822,C 0.2034,E1 1.2678,E2 511.3983} C_DIS
LIN {X 53.5872,Y -128.6506,Z 190,A -57.3298,B 1.1825,C 0.2021,E1 1.2705,E2 510.3647} C_DIS
LIN {X 59.0539,Y -126.2362,Z 190,A -54.9995,B 1.183,C 0.1992,E1 1.2764,E2 508.0511} C_DIS
LIN {X 61.7796,Y -124.9233,Z 190,A -53.7989,B 1.1832,C 0.1975,E1 1.2794,E2 506.8558} C_DIS
LIN {X 65.5601,Y -122.9844,Z 190,A -52.1452,B 1.1836,C 0.1952,E1 1.2835,E2 505.2143} C_DIS
LIN {X 70.0174,Y -120.5019,Z 190,A -50.1852,B 1.1841,C 0.1925,E1 1.2883,E2 503.2726} C_DIS
LIN {X 73.9087,Y -118.1555,Z 190,A -48.4219,B 1.1845,C 0.1898,E1 1.2924,E2 501.5229} C_DIS
LIN {X 77.714,Y -115.6884,Z 190,A -46.6603,B 1.185,C 0.187,E1 1.2965,E2 499.7747} C_DIS
LIN {X 81.3156,Y -113.1856,Z 190,A -45.016,B 1.1854,C 0.1845,E1 1.3003,E2 498.1518} C_DIS
LIN {X 84.4599,Y -110.8589,Z 190,A -43.5015,B 1.1857,C 0.1819,E1 1.3036,E2 496.6494} C_DIS
LIN {X 88.009,Y -108.0628,Z 190,A -41.7742,B 1.1862,C 0.1789,E1 1.3074,E2 494.9393} C_DIS
LIN {X 91.503,Y -105.1205,Z 190,A -40.0794,B 1.1866,C 0.1761,E1 1.3109,E2 493.2692} C_DIS
LIN {X 94.6876,Y -102.262,Z 190,A -38.4191,B 1.1871,C 0.173,E1 1.3143,E2 491.6216} C_DIS
LIN {X 97.9821,Y -99.1097,Z 190,A -36.7156,B 1.1875,C 0.17,E1 1.3177,E2 489.941} C_DIS
LIN {X 101.1029,Y -95.9242,Z 190,A -35.0069,B 1.188,C 0.1667,E1 1.321,E2 488.2485} C_DIS
LIN {X 104.1673,Y -92.5873,Z 190,A -33.3202,B 1.1884,C 0.1635,E1 1.3241,E2 486.5854} C_DIS
LIN {X 107.0678,Y -89.2176,Z 190,A -31.6472,B 1.1889,C 0.1602,E1 1.3271,E2 484.9327} C_DIS
LIN {X 109.9327,Y -85.6624,Z 190,A -29.9424,B 1.1893,C 0.1568,E1 1.33,E2 483.2508} C_DIS
LIN {X 112.5713,Y -82.1645,Z 190,A -28.3238,B 1.1897,C 0.1536,E1 1.3327,E2 481.6565} C_DIS
LIN {X 115.0815,Y -78.6094,Z 190,A -26.6941,B 1.1902,C 0.1502,E1 1.3353,E2 480.0477} C_DIS
LIN {X 117.5629,Y -74.8477,Z 190,A -24.5797,B 1.1909,C 0.1442,E1 1.3385,E2 477.8953} C_DIS
LIN {X 120.0965,Y -70.7103,Z 190,A -23.5119,B 1.1909,C 0.1445,E1 1.3399,E2 476.9553} C_DIS
LIN {X 122.5309,Y -66.4035,Z 190,A -21.359,B 1.1916,C 0.1387,E1 1.3428,E2 474.7845} C_DIS
LIN {X 124.324,Y -62.9775,Z 190,A -20.0142,B 1.1919,C 0.136,E1 1.3445,E2 473.4723} C_DIS
LIN {X 126.566,Y -58.3405,Z 190,A -18.0698,B 1.1924,C 0.1316,E1 1.3468,E2 471.5503} C_DIS
LIN {X 128.2349,Y -54.5801,Z 190,A -16.5696,B 1.1927,C 0.1283,E1 1.3485,E2 470.0752} C_DIS
LIN {X 129.4036,Y -51.7437,Z 190,A -15.4209,B 1.193,C 0.1256,E1 1.3496,E2 468.941} C_DIS
LIN {X 130.708,Y -48.3559,Z 190,A -14.0743,B 1.1933,C 0.1225,E1 1.351,E2 467.6134} C_DIS
LIN {X 132.1267,Y -44.3308,Z 190,A -12.6526,B 1.1936,C 0.1198,E1 1.3522,E2 466.2359} C_DIS
LIN {X 132.9024,Y -41.9497,Z 190,A -11.6185,B 1.1939,C 0.117,E1 1.3531,E2 465.2005} C_DIS
LIN {X 133.6566,Y -39.4791,Z 190,A -10.7449,B 1.1941,C 0.1152,E1 1.3538,E2 464.3517} C_DIS
LIN {X 134.6781,Y -35.8388,Z 190,A -9.1054,B 1.1945,C 0.1105,E1 1.355,E2 462.6995} C_DIS
LIN {X 136.7836,Y -26.7053,Z 190,A -5.8701,B 1.1951,C 0.1036,E1 1.3569,E2 459.5455} C_DIS
LIN {X 137.4101,Y -23.2638,Z 190,A -4.3374,B 1.1955,C 0.099,E1 1.3577,E2 457.9992} C_DIS
LIN {X 138.0826,Y -18.8797,Z 190,A -2.7197,B 1.1958,C 0.0952,E1 1.3583,E2 456.4081} C_DIS
LIN {X 138.58,Y -14.7738,Z 190,A -1.3066,B 1.1961,C 0.0921,E1 1.3587,E2 455.0323} C_DIS
LIN {X 138.9166,Y -11.1874,Z 190,A 0.1117,B 1.1964,C 0.0884,E1 1.3591,E2 453.6215} C_DIS
LIN {X 139.1912,Y -6.9639,Z 190,A 1.6108,B 1.1966,C 0.0849,E1 1.3593,E2 452.1534} C_DIS
LIN {X 139.3373,Y -2.8455,Z 190,A 3.1482,B 1.1969,C 0.0811,E1 1.3594,E2 450.6359} C_DIS
LIN {X 139.3608,Y 1.2317,Z 190,A 4.5589,B 1.1971,C 0.078,E1 1.3594,E2 449.2594} C_DIS
LIN {X 139.274,Y 5.0597,Z 190,A 6.0395,B 1.1973,C 0.0742,E1 1.3593,E2 447.7902} C_DIS
LIN {X 139.0998,Y 8.5988,Z 190,A 7.3414,B 1.1975,C 0.071,E1 1.3591,E2 446.5079} C_DIS
LIN {X 138.8456,Y 12.0274,Z 190,A 8.5416,B 1.1977,C 0.0683,E1 1.3588,E2 445.3348} C_DIS
LIN {X 138.468,Y 15.8039,Z 190,A 9.9123,B 1.1979,C 0.0651,E1 1.3584,E2 443.9882} C_DIS
LIN {X 138.0953,Y 18.7832,Z 190,A 11.1877,B 1.198,C 0.0614,E1 1.358,E2 442.7069} C_DIS
LIN {X 136.7466,Y 26.8986,Z 190,A 14.4306,B 1.1985,C 0.0529,E1 1.3564,E2 439.4805} C_DIS
LIN {X 135.9832,Y 30.52,Z 190,A 15.3576,B 1.1985,C 0.0521,E1 1.3559,E2 438.6298} C_DIS
LIN {X 135.4005,Y 33.0067,Z 190,A 16.4316,B 1.1986,C 0.0491,E1 1.3552,E2 437.5522} C_DIS
LIN {X 134.1281,Y 37.8465,Z 190,A 18.3253,B 1.1988,C 0.0444,E1 1.3538,E2 435.6787} C_DIS
LIN {X 133.0234,Y 41.5697,Z 190,A 19.6794,B 1.1988,C 0.0415,E1 1.3527,E2 434.355} C_DIS
LIN {X 132.0735,Y 44.4904,Z 190,A 20.9375,B 1.199,C 0.0381,E1 1.3516,E2 433.0969} C_DIS
LIN {X 130.5463,Y 48.7877,Z 190,A 22.5671,B 1.1991,C 0.0345,E1 1.3501,E2 431.4979} C_DIS
LIN {X 129.0475,Y 52.6271,Z 190,A 24.0255,B 1.1992,C 0.0314,E1 1.3486,E2 430.0689} C_DIS
LIN {X 127.6647,Y 55.899,Z 190,A 25.6246,B 1.1993,C 0.0268,E1 1.3468,E2 428.4518} C_DIS
LIN {X 126.2811,Y 58.9567,Z 190,A 26.5251,B 1.1993,C 0.0258,E1 1.3458,E2 427.6113} C_DIS
LIN {X 124.8845,Y 61.8583,Z 190,A 27.8619,B 1.1994,C 0.0224,E1 1.3442,E2 426.2724} C_DIS
LIN {X 122.4073,Y 66.6302,Z 190,A 29.8733,B 1.1994,C 0.0178,E1 1.3416,E2 424.2854} C_DIS
LIN {X 120.2438,Y 70.4597,Z 190,A 31.5126,B 1.1995,C 0.0142,E1 1.3393,E2 422.6668} C_DIS
LIN {X 117.8627,Y 74.374,Z 190,A 33.2942,B 1.1995,C 0.0101,E1 1.3367,E2 420.8974} C_DIS
LIN {X 115.8547,Y 77.4648,Z 190,A 34.6039,B 1.1995,C 0.0075,E1 1.3347,E2 419.613} C_DIS
LIN {X 113.1856,Y 81.3156,Z 190,A 36.3061,B 1.1996,C 0.0041,E1 1.332,E2 417.938} C_DIS
LIN {X 110.6576,Y 84.7231,Z 190,A 38.7355,B 1.1996,C -0.0036,E1 1.3277,E2 415.4234} C_DIS
LIN {X 106.1734,Y 90.2791,Z 190,A 40.4005,B 1.1996,C -0.0038,E1 1.325,E2 413.9148} C_DIS
LIN {X 103.7158,Y 93.0922,Z 190,A 41.9822,B 1.1996,C -0.0074,E1 1.3221,E2 412.3274} C_DIS
LIN {X 100.6569,Y 96.3914,Z 190,A 43.6846,B 1.1996,C -0.0108,E1 1.3188,E2 410.6427} C_DIS
LIN {X 97.4885,Y 99.5947,Z 190,A 46.278,B 1.1995,C -0.0184,E1 1.3135,E2 407.9585} C_DIS
LIN {X 91.9723,Y 104.7109,Z 190,A 48.2586,B 1.1995,C -0.0193,E1 1.3096,E2 406.1135} C_DIS
LIN {X 87.9743,Y 108.0912,Z 190,A 50.2144,B 1.1995,C -0.0227,E1 1.3054,E2 404.1813} C_DIS
LIN {X 84.6033,Y 110.7492,Z 190,A 51.8114,B 1.1993,C -0.0253,E1 1.3019,E2 402.6044} C_DIS
LIN {X 81.187,Y 113.2776,Z 190,A 53.5379,B 1.1993,C -0.0285,E1 1.298,E2 400.8805} C_DIS
LIN {X 77.549,Y 115.7985,Z 190,A 55.1531,B 1.1993,C -0.0308,E1 1.2943,E2 399.2896} C_DIS
LIN {X 74.085,Y 118.0451,Z 190,A 56.7671,B 1.1992,C -0.0334,E1 1.2905,E2 397.6857} C_DIS
LIN {X 70.1653,Y 120.4163,Z 190,A 58.536,B 1.1991,C -0.0361,E1 1.2863,E2 395.9306} C_DIS
LIN {X 66.2734,Y 122.6013,Z 190,A 60.2365,B 1.199,C -0.0385,E1 1.2821,E2 394.2461} C_DIS
LIN {X 63.1086,Y 124.2572,Z 190,A 61.8702,B 1.199,C -0.0414,E1 1.278,E2 392.593} C_DIS
LIN {X 59.6866,Y 125.9375,Z 190,A 62.6319,B 1.199,C -0.0404,E1 1.2763,E2 391.9261} C_DIS
LIN {X 56.5495,Y 127.3768,Z 190,A 64.318,B 1.1988,C -0.0436,E1 1.2719,E2 390.2091} C_DIS
LIN {X 53.4995,Y 128.6872,Z 190,A 65.6242,B 1.1988,C -0.0452,E1 1.2686,E2 388.91} C_DIS
LIN {X 50.3362,Y 129.9571,Z 190,A 67.0089,B 1.1987,C -0.047,E1 1.2649,E2 387.5274} C_DIS
LIN {X 46.8748,Y 131.2459,Z 190,A 68.3818,B 1.1987,C -0.0484,E1 1.2614,E2 386.1719} C_DIS
LIN {X 43.2645,Y 132.4817,Z 190,A 70.0199,B 1.1986,C -0.0505,E1 1.257,E2 384.5262} C_DIS
LIN {X 37.0374,Y 134.3543,Z 190,A 72.4427,B 1.1985,C -0.0525,E1 1.2505,E2 382.1331} C_DIS
LIN {X 33.7803,Y 135.2101,Z 190,A 73.753,B 1.1985,C -0.0537,E1 1.2469,E2 380.8317} C_DIS
LIN {X 30.1354,Y 136.0699,Z 190,A 75.629,B 1.1983,C -0.0563,E1 1.2417,E2 378.9171} C_DIS
LIN {X 26.4069,Y 136.8407,Z 190,A 76.528,B 1.1983,C -0.0554,E1 1.2394,E2 378.0956} C_DIS
LIN {X 21.2306,Y 137.7386,Z 190,A 78.8483,B 1.1983,C -0.0577,E1 1.2329,E2 375.7576} C_DIS
LIN {X 17.8376,Y 138.2192,Z 190,A 80.2493,B 1.1982,C -0.0587,E1 1.229,E2 374.358} C_DIS
LIN {X 14.3764,Y 138.6228,Z 190,A 81.548,B 1.1982,C -0.0593,E1 1.2254,E2 373.0751} C_DIS
LIN {X 11.5431,Y 138.8865,Z 190,A 82.772,B 1.1982,C -0.0601,E1 1.222,E2 371.8453} C_DIS
LIN {X 8.1819,Y 139.1255,Z 190,A 84.1943,B 1.1981,C -0.061,E1 1.218,E2 370.4193} C_DIS
LIN {X 3.9901,Y 139.3083,Z 190,A 85.783,B 1.1981,C -0.0614,E1 1.2135,E2 368.8469} C_DIS
LIN {X 0.325,Y 139.3657,Z 190,A 87.2034,B 1.1981,C -0.0617,E1 1.2096,E2 367.4369} C_DIS
LIN {X -3.2962,Y 139.3276,Z 190,A 88.8613,B 1.198,C -0.0627,E1 1.2049,E2 365.7602} C_DIS
LIN {X -7.7281,Y 139.1528,Z 190,A 90.6506,B 1.198,C -0.063,E1 1.1998,E2 363.9757} C_DIS
LIN {X -11.8637,Y 138.8594,Z 190,A 92.2885,B 1.198,C -0.063,E1 1.1953,E2 362.346} C_DIS
LIN {X -18.6397,Y 138.1141,Z 190,A 95.0299,B 1.198,C -0.063,E1 1.1876,E2 359.613} C_DIS
LIN {X -26.1313,Y 136.8933,Z 190,A 97.8589,B 1.198,C -0.062,E1 1.1799,E2 356.8188} C_DIS
LIN {X -30.948,Y 135.8854,Z 190,A 99.959,B 1.198,C -0.0617,E1 1.1741,E2 354.711} C_DIS
LIN {X -33.1582,Y 135.364,Z 190,A 101.1092,B 1.198,C -0.0619,E1 1.1708,E2 353.5367} C_DIS
LIN {X -36.0296,Y 134.6272,Z 190,A 102.4644,B 1.198,C -0.0618,E1 1.1671,E2 352.1665} C_DIS
LIN {X -39.4776,Y 133.6571,Z 190,A 103.8658,B 1.198,C -0.061,E1 1.1633,E2 350.774} C_DIS
LIN {X -42.5824,Y 132.7003,Z 190,A 105.3316,B 1.198,C -0.0606,E1 1.1593,E2 349.2939} C_DIS
LIN {X -46.0661,Y 131.5321,Z 190,A 106.8099,B 1.1981,C -0.0597,E1 1.1554,E2 347.8201} C_DIS
LIN {X -49.1382,Y 130.415,Z 190,A 108.1864,B 1.1981,C -0.0589,E1 1.1518,E2 346.4406} C_DIS
LIN {X -52.7841,Y 128.9842,Z 190,A 110.3007,B 1.1981,C -0.0585,E1 1.1461,E2 344.269} C_DIS
LIN {X -56.4713,Y 127.4118,Z 190,A 111.4051,B 1.1983,C -0.0564,E1 1.1434,E2 343.2282} C_DIS
LIN {X -59.0781,Y 126.2249,Z 190,A 113.0362,B 1.1983,C -0.056,E1 1.1391,E2 341.5457} C_DIS
LIN {X -62.6529,Y 124.4892,Z 190,A 114.3946,B 1.1983,C -0.0541,E1 1.1358,E2 340.22} C_DIS
LIN {X -66.5543,Y 122.4487,Z 190,A 116.4774,B 1.1985,C -0.0526,E1 1.1305,E2 338.1068} C_DIS
LIN {X -71.1126,Y 119.8589,Z 190,A 119.4378,B 1.1985,C -0.0511,E1 1.1231,E2 335.0536} C_DIS
LIN {X -76.0717,Y 116.7744,Z 190,A 121.2348,B 1.1987,C -0.0475,E1 1.119,E2 333.3288} C_DIS
LIN {X -82.4671,Y 112.349,Z 190,A 124.4554,B 1.1988,C -0.0433,E1 1.1116,E2 330.1076} C_DIS
LIN {X -85.1561,Y 110.3251,Z 190,A 126.1117,B 1.1988,C -0.0415,E1 1.1078,E2 328.4204} C_DIS
LIN {X -88.5594,Y 107.6128,Z 190,A 128.0514,B 1.199,C -0.0389,E1 1.1036,E2 326.4641} C_DIS
LIN {X -92.0136,Y 104.6745,Z 190,A 130.0573,B 1.199,C -0.036,E1 1.0993,E2 324.4429} C_DIS
LIN {X -95.1914,Y 101.7929,Z 190,A 131.9791,B 1.1992,C -0.0331,E1 1.0953,E2 322.5035} C_DIS
LIN {X -98.5446,Y 98.5508,Z 190,A 134.0696,B 1.1992,C -0.0298,E1 1.0911,E2 320.3938} C_DIS
LIN {X -101.7556,Y 95.2315,Z 190,A 136.0871,B 1.1993,C -0.0264,E1 1.0871,E2 318.3634} C_DIS
LIN {X -104.6386,Y 92.0543,Z 190,A 137.9949,B 1.1993,C -0.0231,E1 1.0835,E2 316.4396} C_DIS
LIN {X -107.355,Y 88.8708,Z 190,A 139.8538,B 1.1995,C -0.0197,E1 1.0802,E2 314.5653} C_DIS
LIN {X -110.01,Y 85.5626,Z 190,A 142.7052,B 1.1995,C -0.0163,E1 1.0751,E2 311.5812} C_DIS
LIN {X -113.9448,Y 80.2478,Z 190,A 144.8088,B 1.1995,C -0.0105,E1 1.0717,E2 309.5542} C_DIS
LIN {X -116.5675,Y 76.3886,Z 190,A 146.9196,B 1.1996,C -0.0062,E1 1.0684,E2 307.4214} C_DIS
LIN {X -119.0184,Y 72.5114,Z 190,A 149.2826,B 1.1996,C -0.002,E1 1.0648,E2 305.0016} C_DIS
LIN {X -120.8206,Y 69.467,Z 190,A 150.4481,B 1.1996,C 0.0014,E1 1.0633,E2 303.8723} C_DIS
LIN {X -122.5529,Y 66.3632,Z 190,A 152.3278,B 1.1996,C 0.0049,E1 1.0607,E2 301.9425} C_DIS
LIN {X -124.3261,Y 62.9734,Z 190,A 153.9285,B 1.1996,C 0.0087,E1 1.0586,E2 300.3392} C_DIS
LIN {X -125.9961,Y 59.5637,Z 190,A 155.6031,B 1.1996,C 0.0125,E1 1.0566,E2 298.6518} C_DIS
LIN {X -130.1714,Y 49.7851,Z 190,A 160.4583,B 1.1994,C 0.0237,E1 1.0512,E2 293.7399} C_DIS
LIN {X -131.7081,Y 45.5583,Z 190,A 162.4058,B 1.1993,C 0.0285,E1 1.0494,E2 291.7814} C_DIS
LIN {X -132.4596,Y 43.3311,Z 190,A 163.7112,B 1.1993,C 0.0311,E1 1.0482,E2 290.4344} C_DIS
LIN {X -133.371,Y 40.4339,Z 190,A 165.1185,B 1.1991,C 0.0345,E1 1.047,E2 289.0079} C_DIS
LIN {X -134.3583,Y 37.0234,Z 190,A 167.2192,B 1.199,C 0.0386,E1 1.0454,E2 286.8272} C_DIS
LIN {X -135.3295,Y 33.3013,Z 190,A 168.489,B 1.1989,C 0.0427,E1 1.0445,E2 285.5979} C_DIS
LIN {X -136.1084,Y 29.957,Z 190,A 170.0442,B 1.1987,C 0.0466,E1 1.0436,E2 284.0254} C_DIS
LIN {X -136.5978,Y 27.6351,Z 190,A 171.3208,B 1.1986,C 0.0494,E1 1.0428,E2 282.7111} C_DIS
LIN {X -137.3625,Y 23.5495,Z 190,A 173.506,B 1.1984,C 0.0543,E1 1.0417,E2 280.466} C_DIS
LIN {X -138.6668,Y 13.9492,Z 190,A 177.6411,B 1.1978,C 0.0654,E1 1.0403,E2 276.314} C_DIS
LIN {X -138.9605,Y 10.6246,Z 190,A -179.8289,B 1.1976,C 0.0697,E1 1.0397,E2 273.6339} C_DIS
LIN {X -139.2888,Y 4.6782,Z 190,A -177.9611,B 1.1972,C 0.0763,E1 1.0395,E2 271.8437} C_DIS
LIN {X -139.3552,Y -1.773,Z 190,A -175.0399,B 1.1967,C 0.0838,E1 1.0395,E2 268.889} C_DIS
LIN {X -139.2929,Y -4.5428,Z 190,A -173.0206,B 1.1964,C 0.0874,E1 1.0397,E2 266.7542} C_DIS
LIN {X -139.0731,Y -9.0311,Z 190,A -171.2616,B 1.196,C 0.0925,E1 1.04,E2 265.008} C_DIS
LIN {X -138.6599,Y -14.0214,Z 190,A -169.1651,B 1.1956,C 0.0982,E1 1.0405,E2 262.9076} C_DIS
LIN {X -138.31,Y -17.1289,Z 190,A -167.6872,B 1.1953,C 0.1018,E1 1.041,E2 261.4047} C_DIS
LIN {X -137.6543,Y -21.7746,Z 190,A -165.5986,B 1.1948,C 0.1072,E1 1.0419,E2 259.2958} C_DIS
LIN {X -137.1178,Y -24.9297,Z 190,A -164.0503,B 1.1945,C 0.1108,E1 1.0426,E2 257.7169} C_DIS
LIN {X -136.5455,Y -27.8918,Z 190,A -162.6699,B 1.1942,C 0.1142,E1 1.0434,E2 256.3183} C_DIS
LIN {X -135.8609,Y -31.0552,Z 190,A -161.1096,B 1.1938,C 0.1179,E1 1.0443,E2 254.7277} C_DIS
LIN {X -135.0105,Y -34.5667,Z 190,A -159.4749,B 1.1934,C 0.1219,E1 1.0455,E2 253.0734} C_DIS
LIN {X -134.1486,Y -37.7731,Z 190,A -157.8782,B 1.193,C 0.1256,E1 1.0467,E2 251.4459} C_DIS
LIN {X -133.099,Y -41.3227,Z 190,A -156.1516,B 1.1926,C 0.1296,E1 1.0481,E2 249.6921} C_DIS
LIN {X -130.3641,Y -49.2741,Z 190,A -152.3104,B 1.1916,C 0.1386,E1 1.0517,E2 245.7999} C_DIS
LIN {X -129.1321,Y -52.4174,Z 190,A -150.715,B 1.1912,C 0.1421,E1 1.0534,E2 244.1766} C_DIS
LIN {X -127.3382,Y -56.6359,Z 190,A -148.7873,B 1.1906,C 0.1467,E1 1.0555,E2 242.2436} C_DIS
LIN {X -126.3986,Y -58.7026,Z 190,A -147.5799,B 1.1903,C 0.149,E1 1.057,E2 240.9987} C_DIS
LIN {X -124.8523,Y -61.9236,Z 190,A -145.9456,B 1.1899,C 0.1525,E1 1.059,E2 239.3419} C_DIS
LIN {X -123.1409,Y -65.2621,Z 190,A -144.2377,B 1.1894,C 0.1561,E1 1.0613,E2 237.6115} C_DIS
LIN {X -121.1159,Y -68.9497,Z 190,A -142.2124,B 1.1889,C 0.1601,E1 1.0641,E2 235.5455} C_DIS
LIN {X -118.7433,Y -72.9598,Z 190,A -140.1509,B 1.1883,C 0.1644,E1 1.0671,E2 233.4642} C_DIS
LIN {X -116.5536,Y -76.4096,Z 190,A -138.3629,B 1.1878,C 0.168,E1 1.0698,E2 231.6614} C_DIS
LIN {X -114.4809,Y -79.4811,Z 190,A -136.5558,B 1.1873,C 0.1712,E1 1.0728,E2 229.8147} C_DIS
LIN {X -110.6301,Y -84.759,Z 190,A -133.7842,B 1.1865,C 0.1767,E1 1.0774,E2 227.0317} C_DIS
LIN {X -108.4557,Y -87.5241,Z 190,A -132.0652,B 1.1861,C 0.1794,E1 1.0805,E2 225.2742} C_DIS
LIN {X -105.6131,Y -90.9339,Z 190,A -130.0989,B 1.1856,C 0.1829,E1 1.0841,E2 223.2882} C_DIS
LIN {X -103.0269,Y -93.8543,Z 190,A -128.2948,B 1.1852,C 0.1857,E1 1.0875,E2 221.4559} C_DIS
LIN {X -99.8708,Y -97.2063,Z 190,A -125.6396,B 1.1847,C 0.1884,E1 1.0929,E2 218.6917} C_DIS
LIN {X -96.0789,Y -100.9556,Z 190,A -124.0153,B 1.184,C 0.1927,E1 1.096,E2 217.1491} C_DIS
LIN {X -93.3644,Y -103.4714,Z 190,A -122.2317,B 1.1837,C 0.1949,E1 1.0998,E2 215.328} C_DIS
LIN {X -89.3456,Y -106.9605,Z 190,A -119.9159,B 1.1831,C 0.1982,E1 1.1048,E2 212.9939} C_DIS
LIN {X -86.2983,Y -109.4339,Z 190,A -118.1613,B 1.1828,C 0.2004,E1 1.1087,E2 211.219} C_DIS
LIN {X -82.6004,Y -112.251,Z 190,A -116.2358,B 1.1823,C 0.203,E1 1.113,E2 209.2914} C_DIS
LIN {X -79.2025,Y -114.6745,Z 190,A -114.345,B 1.182,C 0.205,E1 1.1174,E2 207.3753} C_DIS
LIN {X -75.4988,Y -117.1462,Z 190,A -112.372,B 1.1816,C 0.207,E1 1.1221,E2 205.3814} C_DIS
LIN {X -71.676,Y -119.5232,Z 190,A -110.4771,B 1.1813,C 0.2091,E1 1.1267,E2 203.48} C_DIS
LIN {X -68.0717,Y -121.6117,Z 190,A -108.7265,B 1.1809,C 0.2108,E1 1.131,E2 201.7236} C_DIS
LIN {X -63.3548,Y -124.1319,Z 190,A -106.7335,B 1.1805,C 0.2134,E1 1.1359,E2 199.76} C_DIS
LIN {X -61.0139,Y -125.301,Z 190,A -105.3532,B 1.1805,C 0.2137,E1 1.1395,E2 198.3354} C_DIS
LIN {X -58.2609,Y -126.6029,Z 190,A -104.0385,B 1.1803,C 0.2147,E1 1.1428,E2 197.0113} C_DIS
LIN {X -55.0578,Y -128.0284,Z 190,A -102.5607,B 1.1801,C 0.2157,E1 1.1467,E2 195.5279} C_DIS
LIN {X -51.3633,Y -129.557,Z 190,A -100.8627,B 1.1799,C 0.2167,E1 1.1511,E2 193.8216} C_DIS
LIN {X -47.5885,Y -130.9886,Z 190,A -99.1292,B 1.1797,C 0.2176,E1 1.1557,E2 192.077} C_DIS
LIN {X -44.2317,Y -132.1597,Z 190,A -97.1527,B 1.1798,C 0.2171,E1 1.1612,E2 190.0248} C_DIS
LIN {X -39.8474,Y -133.5488,Z 190,A -95.7875,B 1.1794,C 0.2193,E1 1.1647,E2 188.7359} C_DIS
LIN {X -35.5575,Y -134.7531,Z 190,A -93.8137,B 1.1794,C 0.2196,E1 1.1701,E2 186.7408} C_DIS
LIN {X -30.9981,Y -135.874,Z 190,A -91.8487,B 1.1793,C 0.22,E1 1.1755,E2 184.77} C_DIS
LIN {X -26.3796,Y -136.8459,Z 190,A -89.9369,B 1.1792,C 0.2204,E1 1.1808,E2 182.8616} C_DIS
LIN {X -22.8263,Y -137.4831,Z 190,A -88.4713,B 1.1792,C 0.2206,E1 1.1848,E2 181.3981} C_DIS
LIN {X -19.5995,Y -137.9802,Z 190,A -87.1022,B 1.1792,C 0.2206,E1 1.1887,E2 180.0245} C_DIS
LIN {X -16.3419,Y -138.4039,Z 190,A -85.8069,B 1.1792,C 0.2206,E1 1.1923,E2 178.7366} C_DIS
LIN {X -12.5874,Y -138.7976,Z 190,A -84.2696,B 1.1792,C 0.2206,E1 1.1966,E2 177.2008} C_DIS
LIN {X -9.0945,Y -139.0692,Z 190,A -82.7349,B 1.1792,C 0.22,E1 1.2009,E2 175.6517} C_DIS
LIN {X -5.1986,Y -139.2685,Z 190,A -81.2035,B 1.1793,C 0.2198,E1 1.2052,E2 174.13} C_DIS
LIN {X -1.9039,Y -139.353,Z 190,A -79.845,B 1.1793,C 0.2194,E1 1.209,E2 172.7703} C_DIS
LIN {X 0.9972,Y -139.3583,Z 190,A -78.8779,B 1.1793,C 0.2197,E1 1.2117,E2 171.8354} C_DIS
Enddeposition()
LIN {X 0.9972,Y -139.3583,Z 190,A -78.8779,B 1.1793,C 0.2197,E1 1.2117,E2 171.8355} C_DIS
Startdeposition()
$VEL.CP = VEL_PRINT
LIN {X 0.4139,Y -140.2641,Z 190,A -79.7015,B 1.2045,C 0.2235,E1 1.2347,E2 172.7633} C_DIS
LIN {X -3.4905,Y -140.2214,Z 190,A -81.1575,B 1.2045,C 0.2235,E1 1.2307,E2 174.1999} C_DIS
LIN {X -7.1307,Y -140.0829,Z 190,A -82.7149,B 1.2044,C 0.2242,E1 1.2263,E2 175.7681} C_DIS
LIN {X -11.0327,Y -139.8317,Z 190,A -84.4364,B 1.2042,C 0.2249,E1 1.2214,E2 177.5086} C_DIS
LIN {X -14.5758,Y -139.5054,Z 190,A -85.7979,B 1.2042,C 0.2247,E1 1.2176,E2 178.8573} C_DIS
LIN {X -18.0326,Y -139.1002,Z 190,A -87.2114,B 1.2042,C 0.2247,E1 1.2136,E2 180.2702} C_DIS
LIN {X -21.6815,Y -138.5784,Z 190,A -88.7058,B 1.2042,C 0.2247,E1 1.2095,E2 181.7636} C_DIS
LIN {X -25.9315,Y -137.8467,Z 190,A -90.5085,B 1.2042,C 0.2246,E1 1.2045,E2 183.573} C_DIS
LIN {X -29.3972,Y -137.1489,Z 190,A -91.7563,B 1.2045,C 0.2237,E1 1.2011,E2 184.7927} C_DIS
LIN {X -34.5276,Y -135.9478,Z 190,A -94.0972,B 1.2045,C 0.2237,E1 1.1946,E2 187.1619} C_DIS
LIN {X -45.1523,Y -132.8002,Z 190,A -98.8223,B 1.2048,C 0.2221,E1 1.1818,E2 191.9175} C_DIS
LIN {X -48.7131,Y -131.5341,Z 190,A -100.2119,B 1.205,C 0.2208,E1 1.1782,E2 193.2851} C_DIS
LIN {X -52.0531,Y -130.2481,Z 190,A -101.8068,B 1.2051,C 0.2201,E1 1.174,E2 194.8996} C_DIS
LIN {X -55.0242,Y -129.0222,Z 190,A -103.2591,B 1.2052,C 0.2195,E1 1.1701,E2 196.3725} C_DIS
LIN {X -58.6035,Y -127.4348,Z 190,A -104.7875,B 1.2055,C 0.218,E1 1.1662,E2 197.8909} C_DIS
LIN {X -62.9865,Y -125.328,Z 190,A -106.8555,B 1.2058,C 0.2164,E1 1.161,E2 199.9711} C_DIS
LIN {X -67.0455,Y -123.2046,Z 190,A -108.9215,B 1.2061,C 0.2149,E1 1.1558,E2 202.0655} C_DIS
LIN {X -71.0885,Y -120.9169,Z 190,A -110.8665,B 1.2064,C 0.213,E1 1.151,E2 204.0177} C_DIS
LIN {X -74.9682,Y -118.5506,Z 190,A -112.834,B 1.2068,C 0.211,E1 1.1463,E2 206.0014} C_DIS
LIN {X -78.5547,Y -116.2052,Z 190,A -114.6841,B 1.2071,C 0.2089,E1 1.1419,E2 207.866} C_DIS
LIN {X -82.1523,Y -113.6904,Z 190,A -116.8155,B 1.2074,C 0.207,E1 1.1369,E2 210.046} C_DIS
LIN {X -84.9089,Y -111.6471,Z 190,A -118.0788,B 1.2078,C 0.2049,E1 1.1341,E2 211.2895} C_DIS
LIN {X -88.3838,Y -108.9171,Z 190,A -120.035,B 1.2082,C 0.2024,E1 1.1298,E2 213.2674} C_DIS
LIN {X -93.4539,Y -104.5985,Z 190,A -123.457,B 1.2088,C 0.1989,E1 1.1224,E2 216.789} C_DIS
LIN {X -97.1367,Y -101.188,Z 190,A -125.6526,B 1.2093,C 0.1956,E1 1.1179,E2 219.0051} C_DIS
LIN {X -100.6328,Y -97.7115,Z 190,A -127.3083,B 1.21,C 0.1916,E1 1.1147,E2 220.6098} C_DIS
LIN {X -103.5676,Y -94.5961,Z 190,A -129.209,B 1.2105,C 0.1886,E1 1.111,E2 222.532} C_DIS
LIN {X -107.2325,Y -90.42,Z 190,A -131.702,B 1.2111,C 0.1844,E1 1.1064,E2 225.0563} C_DIS
LIN {X -113.8723,Y -81.9006,Z 190,A -136.5313,B 1.2124,C 0.1756,E1 1.0981,E2 229.9434} C_DIS
LIN {X -116.4687,Y -78.1641,Z 190,A -138.5576,B 1.213,C 0.1717,E1 1.0948,E2 231.9927} C_DIS
LIN {X -118.7604,Y -74.6358,Z 190,A -140.5202,B 1.2135,C 0.168,E1 1.0918,E2 233.9889} C_DIS
LIN {X -121.1825,Y -70.636,Z 190,A -142.5824,B 1.2141,C 0.1637,E1 1.0889,E2 236.0718} C_DIS
LIN {X -123.3386,Y -66.7999,Z 190,A -144.5799,B 1.2146,C 0.1595,E1 1.0861,E2 238.0964} C_DIS
LIN {X -125.4523,Y -62.7391,Z 190,A -146.6161,B 1.2152,C 0.1551,E1 1.0835,E2 240.155} C_DIS
LIN {X -127.2793,Y -58.9396,Z 190,A -148.5321,B 1.2157,C 0.1509,E1 1.0812,E2 242.097} C_DIS
LIN {X -128.9117,Y -55.2799,Z 190,A -150.421,B 1.2162,C 0.1469,E1 1.079,E2 244.02} C_DIS
LIN {X -130.6179,Y -51.1172,Z 190,A -152.1426,B 1.2168,C 0.1423,E1 1.0773,E2 245.725} C_DIS
LIN {X -131.32,Y -49.2846,Z 190,A -153.651,B 1.217,C 0.1402,E1 1.0757,E2 247.3294} C_DIS
LIN {X -132.6505,Y -45.5841,Z 190,A -155.0357,B 1.2175,C 0.1361,E1 1.0744,E2 248.6834} C_DIS
LIN {X -133.9931,Y -41.4726,Z 190,A -157.0348,B 1.218,C 0.1315,E1 1.0727,E2 250.7134} C_DIS
LIN {X -135.0477,Y -37.8957,Z 190,A -158.6703,B 1.2184,C 0.1274,E1 1.0714,E2 252.3634} C_DIS
LIN {X -135.8523,Y -34.9039,Z 190,A -160.1733,B 1.2188,C 0.124,E1 1.0703,E2 253.8979} C_DIS
LIN {X -136.7305,Y -31.2848,Z 190,A -161.853,B 1.2192,C 0.1199,E1 1.0693,E2 255.5982} C_DIS
LIN {X -137.3331,Y -28.5296,Z 190,A -163.4056,B 1.2195,C 0.1167,E1 1.0683,E2 257.204} C_DIS
LIN {X -138.2021,Y -23.9738,Z 190,A -165.2387,B 1.22,C 0.1115,E1 1.0674,E2 259.028} C_DIS
LIN {X -139.0189,Y -18.6529,Z 190,A -167.8364,B 1.2205,C 0.1054,E1 1.0663,E2 261.6776} C_DIS
LIN {X -139.6115,Y -13.5157,Z 190,A -170.2785,B 1.221,C 0.0994,E1 1.0656,E2 264.1623} C_DIS
LIN {X -140.195,Y -4.4411,Z 190,A -174.2424,B 1.2218,C 0.089,E1 1.065,E2 268.1571} C_DIS
LIN {X -140.2277,Y 3.2633,Z 190,A -177.8462,B 1.2224,C 0.08,E1 1.065,E2 271.819} C_DIS
LIN {X -139.8597,Y 10.6542,Z 190,A 178.5431,B 1.223,C 0.0714,E1 1.0655,E2 275.5042} C_DIS
LIN {X -139.4804,Y 14.808,Z 190,A 176.2246,B 1.2233,C 0.0664,E1 1.0662,E2 277.9004} C_DIS
LIN {X -138.9864,Y 18.9011,Z 190,A 174.1331,B 1.2235,C 0.0616,E1 1.067,E2 280.0427} C_DIS
LIN {X -138.2401,Y 23.7513,Z 190,A 172.432,B 1.2238,C 0.0562,E1 1.0678,E2 281.7041} C_DIS
LIN {X -137.524,Y 27.5911,Z 190,A 170.6161,B 1.224,C 0.0517,E1 1.0687,E2 283.5469} C_DIS
LIN {X -136.8032,Y 30.9668,Z 190,A 169.0533,B 1.2241,C 0.0478,E1 1.0697,E2 285.1282} C_DIS
LIN {X -135.201,Y 37.3476,Z 190,A 166.1721,B 1.2244,C 0.0406,E1 1.0717,E2 288.0321} C_DIS
LIN {X -134.3752,Y 40.2238,Z 190,A 164.6504,B 1.2244,C 0.0372,E1 1.0729,E2 289.5905} C_DIS
LIN {X -133.1772,Y 44.0211,Z 190,A 163.1241,B 1.2246,C 0.033,E1 1.0742,E2 291.1031} C_DIS
LIN {X -132.511,Y 45.9866,Z 190,A 161.8615,B 1.2246,C 0.0306,E1 1.0754,E2 292.4169} C_DIS
LIN {X -130.9067,Y 50.3744,Z 190,A 159.9601,B 1.2248,C 0.0257,E1 1.0773,E2 294.3163} C_DIS
LIN {X -129.9866,Y 52.7018,Z 190,A 157.9954,B 1.2248,C 0.023,E1 1.0795,E2 296.3963} C_DIS
LIN {X -128.0581,Y 57.2278,Z 190,A 156.4547,B 1.2249,C 0.018,E1 1.0811,E2 297.8782} C_DIS
LIN {X -125.7821,Y 62.0706,Z 190,A 154.0772,B 1.2249,C 0.0126,E1 1.084,E2 300.2779} C_DIS
LIN {X -124.2336,Y 65.1145,Z 190,A 152.4361,B 1.225,C 0.0092,E1 1.0862,E2 301.9482} C_DIS
LIN {X -122.1149,Y 69.011,Z 190,A 149.4665,B 1.225,C 0.005,E1 1.0905,E2 305.0563} C_DIS
LIN {X -118.8719,Y 74.4588,Z 190,A 147.4092,B 1.225,C -0.001,E1 1.0934,E2 307.0482} C_DIS
LIN {X -114.8737,Y 80.4903,Z 190,A 143.715,B 1.225,C -0.0074,E1 1.0993,E2 310.8286} C_DIS
LIN {X -112.2374,Y 84.1268,Z 190,A 142.065,B 1.225,C -0.0113,E1 1.102,E2 312.4554} C_DIS
LIN {X -109.0905,Y 88.1688,Z 190,A 139.9204,B 1.225,C -0.0155,E1 1.1058,E2 314.6049} C_DIS
LIN {X -106.3453,Y 91.4612,Z 190,A 137.9717,B 1.225,C -0.0189,E1 1.1093,E2 316.5759} C_DIS
LIN {X -103.4511,Y 94.7228,Z 190,A 135.99,B 1.2249,C -0.0222,E1 1.1131,E2 318.5801} C_DIS
LIN {X -100.2969,Y 98.0563,Z 190,A 133.9651,B 1.2248,C -0.0256,E1 1.1171,E2 320.6214} C_DIS
LIN {X -97.1825,Y 101.1443,Z 190,A 132.0188,B 1.2248,C -0.0287,E1 1.121,E2 322.5847} C_DIS
LIN {X -93.8765,Y 104.2201,Z 190,A 130.0406,B 1.2246,C -0.0317,E1 1.1252,E2 324.5773} C_DIS
LIN {X -90.4782,Y 107.1836,Z 190,A 128.0797,B 1.2246,C -0.0345,E1 1.1294,E2 326.551} C_DIS
LIN {X -86.9775,Y 110.0434,Z 190,A 126.0876,B 1.2245,C -0.0372,E1 1.1338,E2 328.5588} C_DIS
LIN {X -83.4641,Y 112.7314,Z 190,A 124.4278,B 1.2245,C -0.04,E1 1.1374,E2 330.2004} C_DIS
LIN {X -80.7054,Y 114.722,Z 190,A 122.5556,B 1.2244,C -0.0414,E1 1.1419,E2 332.1276} C_DIS
LIN {X -76.1024,Y 117.8261,Z 190,A 120.428,B 1.2242,C -0.0444,E1 1.1468,E2 334.2377} C_DIS
LIN {X -72.4598,Y 120.1002,Z 190,A 118.5104,B 1.2242,C -0.0463,E1 1.1514,E2 336.1731} C_DIS
LIN {X -67.9913,Y 122.6852,Z 190,A 116.2902,B 1.2241,C -0.0485,E1 1.1569,E2 338.4049} C_DIS
LIN {X -63.8739,Y 124.8763,Z 190,A 114.6063,B 1.2241,C -0.0507,E1 1.161,E2 340.0622} C_DIS
LIN {X -60.867,Y 126.3697,Z 190,A 112.9115,B 1.224,C -0.0515,E1 1.1654,E2 341.7934} C_DIS
LIN {X -56.6088,Y 128.3338,Z 190,A 110.6371,B 1.224,C -0.0526,E1 1.1713,E2 344.1077} C_DIS
LIN {X -53.3381,Y 129.7288,Z 190,A 109.322,B 1.2239,C -0.0539,E1 1.1747,E2 345.4064} C_DIS
LIN {X -49.4434,Y 131.2606,Z 190,A 107.6974,B 1.2239,C -0.0552,E1 1.1789,E2 347.0203} C_DIS
LIN {X -46.5707,Y 132.3085,Z 190,A 106.4716,B 1.2238,C -0.056,E1 1.1822,E2 348.2429} C_DIS
LIN {X -43.2317,Y 133.4365,Z 190,A 104.8524,B 1.2238,C -0.0565,E1 1.1866,E2 349.8818} C_DIS
LIN {X -39.8382,Y 134.4881,Z 190,A 103.4681,B 1.2238,C -0.0573,E1 1.1903,E2 351.2577} C_DIS
LIN {X -36.2066,Y 135.5103,Z 190,A 101.9255,B 1.2237,C -0.0579,E1 1.1945,E2 352.7997} C_DIS
LIN {X -33.3815,Y 136.2348,Z 190,A 100.8116,B 1.2237,C -0.0585,E1 1.1975,E2 353.9042} C_DIS
LIN {X -30.1046,Y 136.9962,Z 190,A 99.3475,B 1.2237,C -0.0586,E1 1.2015,E2 355.3779} C_DIS
LIN {X -26.5213,Y 137.7339,Z 190,A 97.7857,B 1.2237,C -0.0588,E1 1.2059,E2 356.9466} C_DIS
LIN {X -23.7688,Y 138.2372,Z 190,A 96.4163,B 1.2237,C -0.0584,E1 1.2097,E2 358.3413} C_DIS
LIN {X -18.0613,Y 139.0965,Z 190,A 94.2599,B 1.2237,C -0.059,E1 1.2157,E2 360.4737} C_DIS
LIN {X -13.8985,Y 139.5747,Z 190,A 92.494,B 1.2237,C -0.0588,E1 1.2206,E2 362.245} C_DIS
LIN {X -10.0704,Y 139.9023,Z 190,A 90.9976,B 1.2237,C -0.0588,E1 1.2248,E2 363.7324} C_DIS
LIN {X -5.936,Y 140.1393,Z 190,A 89.2323,B 1.2237,C -0.0582,E1 1.2298,E2 365.5055} C_DIS
LIN {X -1.841,Y 140.253,Z 190,A 87.6937,B 1.2237,C -0.058,E1 1.2341,E2 367.028} C_DIS
LIN {X 1.783,Y 140.254,Z 190,A 86.1955,B 1.2237,C -0.0574,E1 1.2383,E2 368.5277} C_DIS
LIN {X 5.4828,Y 140.157,Z 190,A 84.7393,B 1.2237,C -0.0569,E1 1.2424,E2 369.9769} C_DIS
LIN {X 9.5073,Y 139.9434,Z 190,A 83.0968,B 1.2237,C -0.0561,E1 1.247,E2 371.6186} C_DIS
LIN {X 13.1609,Y 139.6455,Z 190,A 81.632,B 1.2238,C -0.0553,E1 1.2511,E2 373.0791} C_DIS
LIN {X 17.0077,Y 139.2297,Z 190,A 80.0178,B 1.2238,C -0.0541,E1 1.2556,E2 374.6966} C_DIS
LIN {X 21.1665,Y 138.6581,Z 190,A 78.4952,B 1.2238,C -0.0535,E1 1.2598,E2 376.1966} C_DIS
LIN {X 23.8436,Y 138.2247,Z 190,A 77.2627,B 1.2239,C -0.0522,E1 1.2633,E2 377.4432} C_DIS
LIN {X 27.1106,Y 137.6213,Z 190,A 75.7829,B 1.224,C -0.0506,E1 1.2674,E2 378.9366} C_DIS
LIN {X 30.4295,Y 136.9248,Z 190,A 74.6447,B 1.224,C -0.0501,E1 1.2704,E2 380.0461} C_DIS
LIN {X 34.5092,Y 135.9525,Z 190,A 72.0865,B 1.2242,C -0.0454,E1 1.2777,E2 382.7002} C_DIS
LIN {X 41.8898,Y 133.8651,Z 190,A 69.9768,B 1.2242,C -0.0456,E1 1.283,E2 384.6925} C_DIS
LIN {X 45.606,Y 132.6429,Z 190,A 68.6755,B 1.2242,C -0.0449,E1 1.2864,E2 385.9591} C_DIS
LIN {X 48.9067,Y 131.4616,Z 190,A 67.2283,B 1.2242,C -0.043,E1 1.2902,E2 387.4078} C_DIS
LIN {X 51.7717,Y 130.3615,Z 190,A 65.9571,B 1.2244,C -0.0413,E1 1.2936,E2 388.6809} C_DIS
LIN {X 55.3929,Y 128.8628,Z 190,A 64.6073,B 1.2244,C -0.0401,E1 1.297,E2 390.001} C_DIS
LIN {X 58.2893,Y 127.58,Z 190,A 63.2268,B 1.2244,C -0.0379,E1 1.3005,E2 391.3915} C_DIS
LIN {X 60.8493,Y 126.3781,Z 190,A 62.2047,B 1.2245,C -0.0367,E1 1.3031,E2 392.3979} C_DIS
LIN {X 64.7327,Y 124.4341,Z 190,A 60.4781,B 1.2245,C -0.0342,E1 1.3074,E2 394.1188} C_DIS
LIN {X 68.8097,Y 122.2281,Z 190,A 58.715,B 1.2246,C -0.0317,E1 1.3117,E2 395.8664} C_DIS
LIN {X 72.3163,Y 120.187,Z 190,A 57.108,B 1.2247,C -0.0292,E1 1.3156,E2 397.4673} C_DIS
LIN {X 76.0984,Y 117.8287,Z 190,A 55.2772,B 1.2247,C -0.026,E1 1.3199,E2 399.2992} C_DIS
LIN {X 81.9278,Y 113.8529,Z 190,A 52.742,B 1.2248,C -0.0223,E1 1.3257,E2 401.7934} C_DIS
LIN {X 85.5893,Y 111.1266,Z 190,A 51.031,B 1.2248,C -0.0195,E1 1.3294,E2 403.4861} C_DIS
LIN {X 88.5875,Y 108.7509,Z 190,A 49.5597,B 1.2249,C -0.0168,E1 1.3326,E2 404.9465} C_DIS
LIN {X 92.1015,Y 105.7913,Z 190,A 47.887,B 1.2249,C -0.014,E1 1.3361,E2 406.5949} C_DIS
LIN {X 96.5693,Y 101.7296,Z 190,A 45.4792,B 1.225,C -0.0092,E1 1.3411,E2 408.9958} C_DIS
LIN {X 100.2644,Y 98.0895,Z 190,A 43.6503,B 1.225,C -0.0061,E1 1.3446,E2 410.79} C_DIS
LIN {X 103.2449,Y 94.9471,Z 190,A 42.0949,B 1.225,C -0.0033,E1 1.3476,E2 412.3197} C_DIS
LIN {X 105.9813,Y 91.8837,Z 190,A 40.4532,B 1.225,C 0.0003,E1 1.3506,E2 413.9572} C_DIS
LIN {X 110.0724,Y 86.939,Z 190,A 38.0095,B 1.225,C 0.0054,E1 1.3549,E2 416.3797} C_DIS
LIN {X 113.2302,Y 82.7859,Z 190,A 36.1831,B 1.225,C 0.0088,E1 1.3579,E2 418.1693} C_DIS
LIN {X 115.9269,Y 78.9658,Z 190,A 34.031,B 1.225,C 0.0147,E1 1.3613,E2 420.3513} C_DIS
LIN {X 118.3985,Y 75.2092,Z 190,A 32.7077,B 1.225,C 0.0165,E1 1.3633,E2 421.6121} C_DIS
LIN {X 120.7966,Y 71.2932,Z 190,A 31.006,B 1.2249,C 0.0202,E1 1.3657,E2 423.2927} C_DIS
LIN {X 123.0911,Y 67.2536,Z 190,A 29.3054,B 1.2249,C 0.0239,E1 1.368,E2 424.9693} C_DIS
LIN {X 124.7359,Y 64.1497,Z 190,A 28.0117,B 1.2248,C 0.0268,E1 1.3696,E2 426.2459} C_DIS
LIN {X 126.4287,Y 60.7435,Z 190,A 26.5748,B 1.2247,C 0.0301,E1 1.3713,E2 427.6686} C_DIS
LIN {X 128.3386,Y 56.6008,Z 190,A 24.9233,B 1.2246,C 0.0338,E1 1.3732,E2 429.2942} C_DIS
LIN {X 129.9919,Y 52.6886,Z 190,A 23.4289,B 1.2245,C 0.037,E1 1.3748,E2 430.7589} C_DIS
LIN {X 131.1127,Y 49.8381,Z 190,A 22.2306,B 1.2244,C 0.04,E1 1.376,E2 431.951} C_DIS
LIN {X 132.4086,Y 46.282,Z 190,A 20.9018,B 1.2244,C 0.0429,E1 1.3772,E2 433.2529} C_DIS
LIN {X 133.5949,Y 42.7356,Z 190,A 19.5437,B 1.2242,C 0.0461,E1 1.3784,E2 434.5899} C_DIS
LIN {X 134.6762,Y 39.1959,Z 190,A 17.7489,B 1.224,C 0.0518,E1 1.3798,E2 436.4214} C_DIS
LIN {X 135.8506,Y 34.9106,Z 190,A 16.505,B 1.2239,C 0.0534,E1 1.3807,E2 437.5933} C_DIS
LIN {X 136.7684,Y 31.1191,Z 190,A 14.7637,B 1.2236,C 0.0587,E1 1.3818,E2 439.3542} C_DIS
LIN {X 137.6172,Y 27.132,Z 190,A 13.6364,B 1.2236,C 0.0601,E1 1.3823,E2 440.4133} C_DIS
LIN {X 138.2487,Y 23.6993,Z 190,A 12.2231,B 1.2234,C 0.064,E1 1.383,E2 441.8256} C_DIS
LIN {X 138.9277,Y 19.3228,Z 190,A 10.6015,B 1.2232,C 0.0679,E1 1.3837,E2 443.424} C_DIS
LIN {X 139.4504,Y 15.0873,Z 190,A 9.1757,B 1.223,C 0.0709,E1 1.3841,E2 444.8093} C_DIS
LIN {X 139.728,Y 12.2612,Z 190,A 8.065,B 1.2228,C 0.0738,E1 1.3844,E2 445.9142} C_DIS
LIN {X 139.9889,Y 8.7857,Z 190,A 6.8253,B 1.2226,C 0.0767,E1 1.3846,E2 447.1306} C_DIS
LIN {X 140.1451,Y 5.7897,Z 190,A 5.6982,B 1.2225,C 0.0796,E1 1.3848,E2 448.2455} C_DIS
LIN {X 140.2513,Y 1.9442,Z 190,A 4.2573,B 1.2222,C 0.0832,E1 1.3848,E2 449.6702} C_DIS
LIN {X 140.2481,Y -2.137,Z 190,A 2.817,B 1.222,C 0.0865,E1 1.3848,E2 451.0815} C_DIS
LIN {X 140.1472,Y -5.7346,Z 190,A 1.5045,B 1.2218,C 0.0897,E1 1.3848,E2 452.374} C_DIS
LIN {X 139.9411,Y -9.5388,Z 190,A 0.0361,B 1.2215,C 0.0935,E1 1.3845,E2 453.8318} C_DIS
LIN {X 139.6235,Y -13.3902,Z 190,A -1.3321,B 1.2212,C 0.0966,E1 1.3841,E2 455.1729} C_DIS
LIN {X 139.223,Y -17.064,Z 190,A -2.669,B 1.221,C 0.0998,E1 1.3837,E2 456.4878} C_DIS
LIN {X 138.7018,Y -20.8845,Z 190,A -4.1963,B 1.2206,C 0.1039,E1 1.3831,E2 458.0097} C_DIS
LIN {X 137.9234,Y -25.5297,Z 190,A -5.8651,B 1.2203,C 0.1077,E1 1.3823,E2 459.6456} C_DIS
LIN {X 137.2833,Y -28.7739,Z 190,A -7.0692,B 1.2201,C 0.1105,E1 1.3817,E2 460.8309} C_DIS
LIN {X 136.6194,Y -31.771,Z 190,A -8.6809,B 1.2195,C 0.1161,E1 1.3806,E2 462.4914} C_DIS
LIN {X 135.3935,Y -36.6446,Z 190,A -9.9986,B 1.2195,C 0.1173,E1 1.3797,E2 463.7116} C_DIS
LIN {X 134.4223,Y -40.0631,Z 190,A -11.3072,B 1.2191,C 0.1204,E1 1.3787,E2 465.0018} C_DIS
LIN {X 133.649,Y -42.5665,Z 190,A -12.6199,B 1.2187,C 0.1247,E1 1.3776,E2 466.3481} C_DIS
LIN {X 132.4024,Y -46.2999,Z 190,A -13.779,B 1.2185,C 0.1264,E1 1.3766,E2 467.4475} C_DIS
LIN {X 130.8241,Y -50.587,Z 190,A -15.4277,B 1.2181,C 0.1301,E1 1.375,E2 469.0678} C_DIS
LIN {X 129.6854,Y -53.4421,Z 190,A -16.6363,B 1.2178,C 0.1331,E1 1.3737,E2 470.2709} C_DIS
LIN {X 127.8226,Y -57.7543,Z 190,A -18.5385,B 1.2173,C 0.138,E1 1.3716,E2 472.1722} C_DIS
LIN {X 126.4115,Y -60.7796,Z 190,A -19.6443,B 1.217,C 0.14,E1 1.3703,E2 473.2437} C_DIS
LIN {X 124.426,Y -64.7481,Z 190,A -21.2055,B 1.2167,C 0.1432,E1 1.3683,E2 474.7716} C_DIS
LIN {X 122.8837,Y -67.6329,Z 190,A -22.3884,B 1.2164,C 0.1457,E1 1.3668,E2 475.9343} C_DIS
LIN {X 120.1938,Y -72.3048,Z 190,A -24.6066,B 1.2157,C 0.1512,E1 1.3636,E2 478.1565} C_DIS
LIN {X 118.4698,Y -75.0963,Z 190,A -25.6422,B 1.2155,C 0.1528,E1 1.3621,E2 479.1509} C_DIS
LIN {X 116.0612,Y -78.7673,Z 190,A -27.2954,B 1.215,C 0.1563,E1 1.3596,E2 480.7859} C_DIS
LIN {X 113.3838,Y -82.5753,Z 190,A -29.0047,B 1.2146,C 0.1598,E1 1.3569,E2 482.4698} C_DIS
LIN {X 110.756,Y -86.0675,Z 190,A -30.6114,B 1.2142,C 0.1629,E1 1.3542,E2 484.0529} C_DIS
LIN {X 107.9971,Y -89.5047,Z 190,A -32.2956,B 1.2137,C 0.1664,E1 1.3512,E2 485.7222} C_DIS
LIN {X 104.9943,Y -93.009,Z 190,A -33.9939,B 1.2133,C 0.1696,E1 1.3481,E2 487.3957} C_DIS
LIN {X 101.9901,Y -96.2937,Z 190,A -35.6749,B 1.2128,C 0.1729,E1 1.345,E2 489.0588} C_DIS
LIN {X 98.7746,Y -99.5894,Z 190,A -37.4102,B 1.2123,C 0.1761,E1 1.3416,E2 490.775} C_DIS
LIN {X 95.5707,Y -102.6679,Z 190,A -39.0826,B 1.2119,C 0.1792,E1 1.3382,E2 492.4286} C_DIS
LIN {X 92.1651,Y -105.7358,Z 190,A -40.8198,B 1.2114,C 0.1823,E1 1.3346,E2 494.148} C_DIS
LIN {X 88.5994,Y -108.7412,Z 190,A -42.585,B 1.211,C 0.1853,E1 1.3308,E2 495.8949} C_DIS
LIN {X 84.9352,Y -111.627,Z 190,A -44.3147,B 1.2105,C 0.188,E1 1.3271,E2 497.601} C_DIS
LIN {X 81.5952,Y -114.0907,Z 190,A -45.8997,B 1.2101,C 0.1906,E1 1.3235,E2 499.1716} C_DIS
LIN {X 78.1068,Y -116.5069,Z 190,A -47.5506,B 1.2097,C 0.1933,E1 1.3197,E2 500.8121} C_DIS
LIN {X 74.5211,Y -118.8328,Z 190,A -49.1986,B 1.2093,C 0.1959,E1 1.3158,E2 502.4474} C_DIS
LIN {X 70.6756,Y -121.1594,Z 190,A -50.7601,B 1.209,C 0.1976,E1 1.3121,E2 503.9709} C_DIS
LIN {X 65.0942,Y -124.2443,Z 190,A -53.2458,B 1.2084,C 0.2012,E1 1.3061,E2 506.4413} C_DIS
LIN {X 62.1187,Y -125.7583,Z 190,A -55.5168,B 1.2074,C 0.2075,E1 1.3,E2 508.8431} C_DIS
LIN {X 55.1571,Y -128.9647,Z 190,A -57.5804,B 1.2074,C 0.207,E1 1.2951,E2 510.7564} C_DIS
LIN {X 51.0871,Y -130.6297,Z 190,A -59.1771,B 1.2072,C 0.2085,E1 1.291,E2 512.3255} C_DIS
LIN {X 47.906,Y -131.8297,Z 190,A -60.5542,B 1.2069,C 0.2102,E1 1.2873,E2 513.7018} C_DIS
LIN {X 44.6698,Y -132.9612,Z 190,A -61.6789,B 1.2069,C 0.2107,E1 1.2845,E2 514.7876} C_DIS
LIN {X 39.882,Y -134.4753,Z 190,A -63.8633,B 1.2063,C 0.2136,E1 1.2786,E2 516.9927} C_DIS
LIN {X 36.1742,Y -135.5189,Z 190,A -65.3178,B 1.2061,C 0.2148,E1 1.2746,E2 518.431} C_DIS
LIN {X 33.4918,Y -136.2082,Z 190,A -66.4248,B 1.2059,C 0.2158,E1 1.2716,E2 519.5353} C_DIS
LIN {X 28.4566,Y -137.3479,Z 190,A -68.6139,B 1.2055,C 0.2181,E1 1.2656,E2 521.7374} C_DIS
LIN {X 23.8205,Y -138.2286,Z 190,A -70.2827,B 1.2054,C 0.2187,E1 1.2611,E2 523.3698} C_DIS
LIN {X 20.6066,Y -138.7443,Z 190,A -71.6395,B 1.2052,C 0.2198,E1 1.2573,E2 524.7313} C_DIS
LIN {X 16.9082,Y -139.2416,Z 190,A -73.084,B 1.205,C 0.2206,E1 1.2533,E2 526.1651} C_DIS
Enddeposition()
END
